THE SOFTWARE IS PROVIDED "AS IS", WITHOUT WARRANTY OF ANY KIND, EXPRESS OR 
IMPLIED, INCLUDING BUT NOT LIMITED TO THE WARRANTIES OF MERCHANTABILITY, 
FITNESS FOR A PARTICULAR PURPOSE AND NONINFRINGEMENT. IN NO EVENT SHALL THE 
AUTHORS OR COPYRIGHT HOLDERS BE LIABLE FOR ANY CLAIM, DAMAGES OR OTHER 
LIABILITY, WHETHER IN AN ACTION OF CONTRACT, TORT OR OTHERWISE, ARISING FROM, 
OUT OF OR IN CONNECTION WITH THE SOFTWARE OR THE USE OR OTHER DEALINGS 
IN THE SOFTWARE.
*)
fin := FALSE;
                    
END_ACTION
END_PROGRAM

(* Moves VG in x, y and z axis Copyright (c) 2019 Manuel Goester, Michael Witt, Klaus Kammerer Institute of Databases and Information Systems, Ulm University, Germany Permission is hereby granted, free of charge, to any person obtaining a copy of this software and associated documentation files (the "Software"), to deal in the Software without restriction, including without limitation the rights to use, copy, modify, merge, publish, distribute, sublicense, and/or sell copies of the Software, and to permit persons to whom the Software is furnished to do so, subject to the following conditions: The above copyright notice and this permission notice shall be included in all copies or substantial portions of the Software. THE SOFTWARE IS PROVIDED "AS IS", WITHOUT WARRANTY OF ANY KIND, EXPRESS OR IMPLIED, INCLUDING BUT NOT LIMITED TO THE WARRANTIES OF MERCHANTABILITY, FITNESS FOR A PARTICULAR PURPOSE AND NONINFRINGEMENT. IN NO EVENT SHALL THE AUTHORS OR COPYRIGHT HOLDERS BE LIABLE FOR ANY CLAIM, DAMAGES OR OTHER LIABILITY, WHETHER IN AN ACTION OF CONTRACT, TORT OR OTHERWISE, ARISING FROM, OUT OF OR IN CONNECTION WITH THE SOFTWARE OR THE USE OR OTHER DEALINGS IN THE SOFTWARE. *)
FUNCTION_BLOCK VG_MOVE
  VAR_INPUT
    x : INT;  (* distance VG will go forward (positive value) or backward (negative value) *)
    y : INT;  (* distance VG will go down (positive value) or up (negative value) *)
    z : INT;  (* distance VG will go counter clockwise (positive value) or clockwise (negative value) *)
  END_VAR
  VAR
    xFin : BOOL := FALSE;  (* finish flags *)
    yFin : BOOL := FALSE;
    zFin : BOOL := FALSE;
    fin : BOOL := FALSE;
    xAlreadyCounted : BOOL := FALSE;  (* true, if an impulse coming from the motor has been already counted *)
    yAlreadyCounted : BOOL := FALSE;
    zAlreadyCounted : BOOL := FALSE;
    cX : INT := 0;  (* counters *)
    cY : INT := 0;
    cZ : INT := 0;
  END_VAR

                  fin := FALSE;

// X AXIS (Forward/Backward)
IF x < 0 THEN
	// drive backward
	IF cX = x THEN
		// if counter reached demanded position, we're done
		VG.mHorizontalBackward := FALSE;
		xFin := TRUE;
	ELSE
		xFin := FALSE;
		IF cX > x THEN
			VG.mHorizontalBackward := TRUE;
			IF VG.encHorizontal AND NOT(xAlreadyCounted) THEN
				// update local counter
				cX := cX - 1;
				// update global counter
				VG.cX := VG.cX - 1;
				xAlreadyCounted := TRUE;
			ELSIF NOT(VG.encHorizontal) THEN
				xAlreadyCounted := FALSE;
			END_IF
		END_IF
	END_IF
ELSE
	// x >= 0
	// drive forward
	IF cX = x THEN
		// if counter reached demanded position, we're done
		VG.mHorizontalForward := FALSE;
		xFin := TRUE;
	ELSE
		xFin := FALSE;
		IF cX < x THEN
			VG.mHorizontalForward := TRUE;
			IF VG.encHorizontal AND NOT(xAlreadyCounted) THEN
				// update local counter
				cX := cX + 1;
				// update global counter
				VG.cX := VG.cX + 1;
				xAlreadyCounted := TRUE;
			ELSIF NOT(VG.encHorizontal) THEN
				xAlreadyCounted := FALSE;
			END_IF
		END_IF
	END_IF
END_IF

// Y AXIS (Up/Down)
IF y < 0 THEN
	// drive up
	IF cY = y THEN
		// if counter reached demanded position, we're done
		VG.mVerticalUp := FALSE;
		yFin := TRUE;
	ELSE
		yFin := FALSE;
		IF cY > y THEN
			VG.mVerticalUp := TRUE;
			IF VG.encVertical AND NOT(yAlreadyCounted) THEN
				// update local counter
				cY := cY - 1;
				// update global counter
				VG.cY := VG.cY - 1;
				yAlreadyCounted := TRUE;
			ELSIF NOT(VG.encVertical) THEN
				yAlreadyCounted := FALSE;
			END_IF
		END_IF
	END_IF
ELSE
	// y >= 0
	// drive down
	IF cY = y THEN
		// if counter reached demanded position, we're done
		VG.mVerticalDown := FALSE;
	yFin := TRUE;
	ELSE
		yFin := FALSE;
		IF cY < y THEN
			VG.mVerticalDown := TRUE;
			IF VG.encVertical AND NOT(yAlreadyCounted) THEN
				// update local counter
				cY := cY + 1;
				// update global counter
				VG.cY := VG.cY + 1;
				yAlreadyCounted := TRUE;
			ELSIF NOT(VG.encVertical) THEN
				yAlreadyCounted := FALSE;
			END_IF
		END_IF
	END_IF
END_IF

// Z AXIS (Rotation)
IF z < 0 THEN
	// drive clockwise
	IF cZ = z THEN
		// if counter reached demanded position, we're done
		VG.mRotationClockwise := FALSE;
		zFin := TRUE;
	ELSE
		zFin := FALSE;
		IF cZ > z THEN
			VG.mRotationClockwise := TRUE;
			IF VG.encRotation AND NOT(zAlreadyCounted) THEN
				// update local counter
				cZ := cZ - 1;
				// update global counter
				VG.cZ := VG.cZ - 1;
				zAlreadyCounted := TRUE;
			ELSIF NOT(VG.encRotation) THEN
				zAlreadyCounted := FALSE;
			END_IF
		END_IF
	END_IF
ELSE
	// z >= 0
	// drive counter clockwise
	IF cZ = z THEN
		// if counter reached demanded position, we're done
		VG.mRotationCClockwise := FALSE;
		zFin := TRUE;
	ELSE
		zFin := FALSE;
		IF cZ < z THEN
			VG.mRotationCClockwise := TRUE;
			IF VG.encRotation AND NOT(zAlreadyCounted) THEN
				// update local counter
				cZ := cZ + 1;
				// update global counter
				VG.cZ := VG.cZ + 1;
				zAlreadyCounted := TRUE;
			ELSIF NOT(VG.encRotation) THEN
				zAlreadyCounted := FALSE;
			END_IF
		END_IF
	END_IF
END_IF

// if all axes are finsihed, we're done
IF xFin AND yFin AND zFin THEN
	// reset local counters
	cX := 0;
	cY := 0;
	cZ := 0;
	fin := TRUE;
	RETURN;
END_IF
                
END_FUNCTION_BLOCK

PROGRAM HR_MULTI_MODE
  VAR
    fin : BOOL;
    hr_get : HR_GET_W;
    hr_store : HR_STORE_W;
    hr_put_w_on_conveyor : HR_PUT_W_ON_CONVEYOR;
    calibrateYAxis : INT := 0;  (* for GET_W calibrate y axis of rack every 3th workpiece *)
    calibarteYAxisCounted : BOOL := FALSE;
    step : INT := 1;
    timer : TON;
  END_VAR

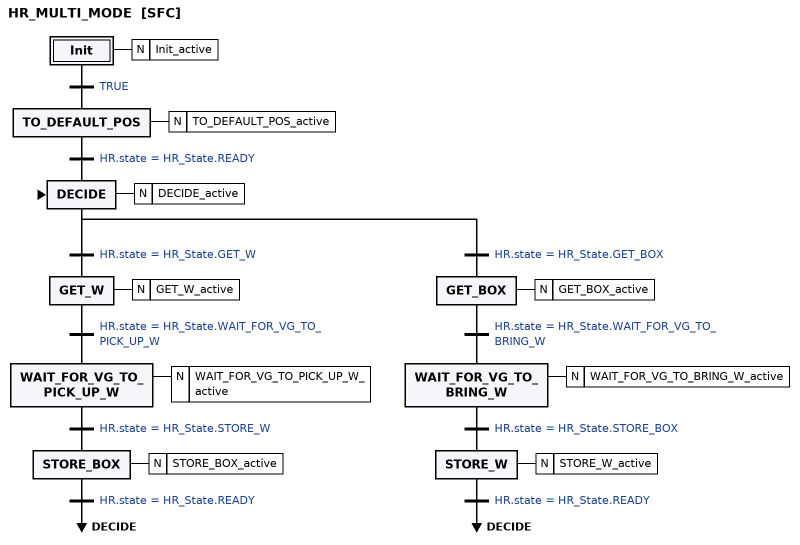
INITIAL_STEP Init:
  Init_active(N);
END_STEP
TRANSITION FROM Init TO TO_DEFAULT_POS
  := TRUE;
END_TRANSITION
STEP TO_DEFAULT_POS:
  TO_DEFAULT_POS_active(N);
END_STEP
TRANSITION FROM TO_DEFAULT_POS TO DECIDE
  := HR.state = HR_State.READY;
END_TRANSITION
STEP DECIDE:
  DECIDE_active(N);
END_STEP
TRANSITION FROM DECIDE TO GET_W
  := HR.state = HR_State.GET_W;
END_TRANSITION
TRANSITION FROM DECIDE TO GET_BOX
  := HR.state = HR_State.GET_BOX;
END_TRANSITION
STEP GET_W:
  GET_W_active(N);
END_STEP
TRANSITION FROM GET_W TO WAIT_FOR_VG_TO_PICK_UP_W
  := HR.state = HR_State.WAIT_FOR_VG_TO_PICK_UP_W;
END_TRANSITION
STEP WAIT_FOR_VG_TO_PICK_UP_W:
  WAIT_FOR_VG_TO_PICK_UP_W_active(N);
END_STEP
TRANSITION FROM WAIT_FOR_VG_TO_PICK_UP_W TO STORE_BOX
  := HR.state = HR_State.STORE_W;
END_TRANSITION
STEP STORE_BOX:
  STORE_BOX_active(N);
END_STEP
TRANSITION FROM STORE_BOX TO DECIDE
  := HR.state = HR_State.READY;
END_TRANSITION
STEP GET_BOX:
  GET_BOX_active(N);
END_STEP
TRANSITION FROM GET_BOX TO WAIT_FOR_VG_TO_BRING_W
  := HR.state = HR_State.WAIT_FOR_VG_TO_BRING_W;
END_TRANSITION
STEP WAIT_FOR_VG_TO_BRING_W:
  WAIT_FOR_VG_TO_BRING_W_active(N);
END_STEP
TRANSITION FROM WAIT_FOR_VG_TO_BRING_W TO STORE_W
  := HR.state = HR_State.STORE_BOX;
END_TRANSITION
STEP STORE_W:
  STORE_W_active(N);
END_STEP
TRANSITION FROM STORE_W TO DECIDE
  := HR.state = HR_State.READY;
END_TRANSITION

ACTION STORE_BOX_active:
                      (*
Copyright (c) 2019 Manuel Goester, Michael Witt, Klaus Kammerer
Institute of Databases and Information Systems, Ulm University, Germany

Permission is hereby granted, free of charge, to any person obtaining a copy 
of this software and associated documentation files (the "Software"), to deal 
in the Software without restriction, including without limitation the rights 
to use, copy, modify, merge, publish, distribute, sublicense, and/or sell 
copies of the Software, and to permit persons to whom the Software is 
furnished to do so, subject to the following conditions:

The above copyright notice and this permission notice shall be included in 
all copies or substantial portions of the Software.

THE SOFTWARE IS PROVIDED "AS IS", WITHOUT WARRANTY OF ANY KIND, EXPRESS OR 
IMPLIED, INCLUDING BUT NOT LIMITED TO THE WARRANTIES OF MERCHANTABILITY, 
FITNESS FOR A PARTICULAR PURPOSE AND NONINFRINGEMENT. IN NO EVENT SHALL THE 
AUTHORS OR COPYRIGHT HOLDERS BE LIABLE FOR ANY CLAIM, DAMAGES OR OTHER 
LIABILITY, WHETHER IN AN ACTION OF CONTRACT, TORT OR OTHERWISE, ARISING FROM, 
OUT OF OR IN CONNECTION WITH THE SOFTWARE OR THE USE OR OTHER DEALINGS 
IN THE SOFTWARE.
*)
IF NOT fin THEN
	// store box in rack
	hr_store(w := HR.currW);
	fin := hr_store.fin;
ELSE
	fin := FALSE;
	HR.state := HR_State.READY;
END_IF
                    
END_ACTION

ACTION GET_W_active:
                      (*
Copyright (c) 2019 Manuel Goester, Michael Witt, Klaus Kammerer
Institute of Databases and Information Systems, Ulm University, Germany

Permission is hereby granted, free of charge, to any person obtaining a copy 
of this software and associated documentation files (the "Software"), to deal 
in the Software without restriction, including without limitation the rights 
to use, copy, modify, merge, publish, distribute, sublicense, and/or sell 
copies of the Software, and to permit persons to whom the Software is 
furnished to do so, subject to the following conditions:

The above copyright notice and this permission notice shall be included in 
all copies or substantial portions of the Software.

THE SOFTWARE IS PROVIDED "AS IS", WITHOUT WARRANTY OF ANY KIND, EXPRESS OR 
IMPLIED, INCLUDING BUT NOT LIMITED TO THE WARRANTIES OF MERCHANTABILITY, 
FITNESS FOR A PARTICULAR PURPOSE AND NONINFRINGEMENT. IN NO EVENT SHALL THE 
AUTHORS OR COPYRIGHT HOLDERS BE LIABLE FOR ANY CLAIM, DAMAGES OR OTHER 
LIABILITY, WHETHER IN AN ACTION OF CONTRACT, TORT OR OTHERWISE, ARISING FROM, 
OUT OF OR IN CONNECTION WITH THE SOFTWARE OR THE USE OR OTHER DEALINGS 
IN THE SOFTWARE.
*)
// increment y calibration counter
IF NOT(calibarteYAxisCounted) THEN
	calibrateYAxis := calibrateYAxis + 1;
	calibarteYAxisCounted := TRUE;
END_IF

IF calibrateYAxis >= 3 THEN
	// calibrate y axis
	IF NOT(HR.sVertical) THEN
		HR.mVerticalUp := TRUE;
	ELSE
		Hr.mVerticalUp := FALSE;
		Hr.cY := 0;
		calibrateYAxis := 0;
	END_IF
ELSE
	CASE step OF
		1:
			// get w from rack
			IF NOT fin THEN
				hr_get(w:= HR.currW);
				fin := hr_get.fin;
			ELSE
				fin := FALSE;
				step := step + 1;
			END_IF
		2:
			// put w on conveyor
			hr_put_w_on_conveyor(w := HR.currW);
			fin := hr_put_w_on_conveyor.fin;	
			IF fin THEN
				step := step + 1;
				fin := FALSE;
			END_IF
		3:
			// bring it to VG in conveyor
			IF HR.lbOut THEN
				HR.mCbForward := TRUE;
			ELSE
				// start 1 sec timer to drive conveyor 1 sec longer to be sure that box is at outside pos
				timer(IN:= TRUE, PT := T#1S);
				IF NOT(timer.Q = FALSE AND timer.IN) THEN
					timer(IN:= FALSE);
					HR.mCbForward := FALSE;
					step := step + 1; 
				END_IF
			END_IF
		4:
			// finished
			step := 1;
			HR.state := HR_State.WAIT_FOR_VG_TO_PICK_UP_W;
			calibarteYAxisCounted := FALSE;
			// bend VG pointers to current workpiece of HR
			VG.bIdx := TC.currBatchJobIdx;
			VG.wIdx := TC.batchJobQueue.batchJobs[TC.currBatchJobIdx].nextNotProcessedIdx;
			VG.currW := TC.batchJobQueue.batchJobs[VG.bIdx].workpieces[VG.wIdx];
	END_CASE
END_IF


                    
END_ACTION

ACTION WAIT_FOR_VG_TO_PICK_UP_W_active:
                      (*
Copyright (c) 2019 Manuel Goester, Michael Witt, Klaus Kammerer
Institute of Databases and Information Systems, Ulm University, Germany

Permission is hereby granted, free of charge, to any person obtaining a copy 
of this software and associated documentation files (the "Software"), to deal 
in the Software without restriction, including without limitation the rights 
to use, copy, modify, merge, publish, distribute, sublicense, and/or sell 
copies of the Software, and to permit persons to whom the Software is 
furnished to do so, subject to the following conditions:

The above copyright notice and this permission notice shall be included in 
all copies or substantial portions of the Software.

THE SOFTWARE IS PROVIDED "AS IS", WITHOUT WARRANTY OF ANY KIND, EXPRESS OR 
IMPLIED, INCLUDING BUT NOT LIMITED TO THE WARRANTIES OF MERCHANTABILITY, 
FITNESS FOR A PARTICULAR PURPOSE AND NONINFRINGEMENT. IN NO EVENT SHALL THE 
AUTHORS OR COPYRIGHT HOLDERS BE LIABLE FOR ANY CLAIM, DAMAGES OR OTHER 
LIABILITY, WHETHER IN AN ACTION OF CONTRACT, TORT OR OTHERWISE, ARISING FROM, 
OUT OF OR IN CONNECTION WITH THE SOFTWARE OR THE USE OR OTHER DEALINGS 
IN THE SOFTWARE.
*)
IF VG.state = VG_State.TO_FUR_PUT_W OR VG.state = VG_State.TO_EJECT THEN
	HR.state := HR_State.STORE_W;
	HR.decidedToTakeANewW := FALSE;
END_IF
                    
END_ACTION

ACTION GET_BOX_active:
                      (*
Copyright (c) 2019 Manuel Goester, Michael Witt, Klaus Kammerer
Institute of Databases and Information Systems, Ulm University, Germany

Permission is hereby granted, free of charge, to any person obtaining a copy 
of this software and associated documentation files (the "Software"), to deal 
in the Software without restriction, including without limitation the rights 
to use, copy, modify, merge, publish, distribute, sublicense, and/or sell 
copies of the Software, and to permit persons to whom the Software is 
furnished to do so, subject to the following conditions:

The above copyright notice and this permission notice shall be included in 
all copies or substantial portions of the Software.

THE SOFTWARE IS PROVIDED "AS IS", WITHOUT WARRANTY OF ANY KIND, EXPRESS OR 
IMPLIED, INCLUDING BUT NOT LIMITED TO THE WARRANTIES OF MERCHANTABILITY, 
FITNESS FOR A PARTICULAR PURPOSE AND NONINFRINGEMENT. IN NO EVENT SHALL THE 
AUTHORS OR COPYRIGHT HOLDERS BE LIABLE FOR ANY CLAIM, DAMAGES OR OTHER 
LIABILITY, WHETHER IN AN ACTION OF CONTRACT, TORT OR OTHERWISE, ARISING FROM, 
OUT OF OR IN CONNECTION WITH THE SOFTWARE OR THE USE OR OTHER DEALINGS 
IN THE SOFTWARE.
*)
CASE step OF
	1:
		IF NOT fin THEN
			hr_get(w:= HR.currW);
			fin := hr_get.fin;
		ELSE
			step := step + 1;
			fin := FALSE;
		END_IF
	2:
		// put w on conveyor
		hr_put_w_on_conveyor(w := HR.currW);
		fin := hr_put_w_on_conveyor.fin;	
		IF fin THEN
			step := step + 1;
			fin := FALSE;
		END_IF
	3:
		// bring it to VG in conveyor
		IF HR.lbOut THEN
			HR.mCbForward := TRUE;
		ELSE
			// start 1 sec timer to drive conveyor 1 sec longer to be sure that box is at outside pos
			timer(IN:= TRUE, PT := T#1S);
			IF NOT(timer.Q = FALSE AND timer.IN) THEN
				timer(IN:= FALSE);
				HR.mCbForward := FALSE;
				step := step + 1; 
			END_IF
		END_IF
	4:
		// finished
		step := 1;
		HR.state := HR_State.WAIT_FOR_VG_TO_BRING_W;
END_CASE
                    
END_ACTION

ACTION DECIDE_active:
                      (*
Copyright (c) 2019 Manuel Goester, Michael Witt, Klaus Kammerer
Institute of Databases and Information Systems, Ulm University, Germany

Permission is hereby granted, free of charge, to any person obtaining a copy 
of this software and associated documentation files (the "Software"), to deal 
in the Software without restriction, including without limitation the rights 
to use, copy, modify, merge, publish, distribute, sublicense, and/or sell 
copies of the Software, and to permit persons to whom the Software is 
furnished to do so, subject to the following conditions:

The above copyright notice and this permission notice shall be included in 
all copies or substantial portions of the Software.

THE SOFTWARE IS PROVIDED "AS IS", WITHOUT WARRANTY OF ANY KIND, EXPRESS OR 
IMPLIED, INCLUDING BUT NOT LIMITED TO THE WARRANTIES OF MERCHANTABILITY, 
FITNESS FOR A PARTICULAR PURPOSE AND NONINFRINGEMENT. IN NO EVENT SHALL THE 
AUTHORS OR COPYRIGHT HOLDERS BE LIABLE FOR ANY CLAIM, DAMAGES OR OTHER 
LIABILITY, WHETHER IN AN ACTION OF CONTRACT, TORT OR OTHERWISE, ARISING FROM, 
OUT OF OR IN CONNECTION WITH THE SOFTWARE OR THE USE OR OTHER DEALINGS 
IN THE SOFTWARE.
*)

// if sl positions free or if not free if workpiece will not be ejected 
// AND VG is not storing
// AND HR does not already decided to take a new workpiece
// THEN 
IF ((SL.lbRed AND SL.lbWhite AND SL.lbBlue) OR (SL.currW.format.ejectEnabled AND NOT(SL.currW.state = W_State.NULL))) AND NOT(VG.storeW) AND NOT(decidedToTakeANewW) THEN
	HR.bIdx := 0;
	HR.wIdx := 0;
	HR.currW := TC.nullW;
	HR.decidedToTakeANewW := TRUE;
	VG.storeW := FALSE;
ELSIF HR.decidedToTakeANewW THEN
	// get new w out of rack
	IF TC.state = TC_state.W_LOADED THEN
		// set pointers to make sure that they are set
		Hr.bIdx := TC.currBatchJobIdx;
		Hr.wIdx := TC.batchJobQueue.batchJobs[TC.currBatchJobIdx].nextNotProcessedIdx;
		HR.currW := TC.batchJobQueue.batchJobs[Hr.bIdx].workpieces[Hr.wIdx];
		// workpiece is loaded, start production
		HR.state := HR_State.GET_W;
		// signalise that production starts
		TC.state := TC_State.WAIT_UNTIL_W_FINISHED;
	ELSE
		// no workpiece loaded, load it now
		TC.state := TC_State.LOAD_NEXT_W;
	END_IF
ELSE
	// prevent misconduct when a workpiece is still lying in one of the three spots at SL, although the application got reset
	IF NOT(VG.bIdx = 0) THEN
		// get empty box out of rack
		// set workpiece to get the right box from rack
		IF NOT(SL.lbWhite) OR NOT(SL.lbRed) OR NOT(SL.lbBlue) THEN
			HR.bIdx := SL.bIdx;
			HR.wIdx := SL.wIdx;
			HR.currW := SL.currW;
		ELSE
			HR.bIdx := VG.bIdx;
			HR.wIdx := VG.wIdx;
			HR.currW := VG.currW;
		END_IF
		HR.state := HR_State.GET_BOX;
		// reset flag
		VG.storeW := FALSE;
		END_IF
END_IF
                    
END_ACTION

ACTION STORE_W_active:
                      (*
Copyright (c) 2019 Manuel Goester, Michael Witt, Klaus Kammerer
Institute of Databases and Information Systems, Ulm University, Germany

Permission is hereby granted, free of charge, to any person obtaining a copy 
of this software and associated documentation files (the "Software"), to deal 
in the Software without restriction, including without limitation the rights 
to use, copy, modify, merge, publish, distribute, sublicense, and/or sell 
copies of the Software, and to permit persons to whom the Software is 
furnished to do so, subject to the following conditions:

The above copyright notice and this permission notice shall be included in 
all copies or substantial portions of the Software.

THE SOFTWARE IS PROVIDED "AS IS", WITHOUT WARRANTY OF ANY KIND, EXPRESS OR 
IMPLIED, INCLUDING BUT NOT LIMITED TO THE WARRANTIES OF MERCHANTABILITY, 
FITNESS FOR A PARTICULAR PURPOSE AND NONINFRINGEMENT. IN NO EVENT SHALL THE 
AUTHORS OR COPYRIGHT HOLDERS BE LIABLE FOR ANY CLAIM, DAMAGES OR OTHER 
LIABILITY, WHETHER IN AN ACTION OF CONTRACT, TORT OR OTHERWISE, ARISING FROM, 
OUT OF OR IN CONNECTION WITH THE SOFTWARE OR THE USE OR OTHER DEALINGS 
IN THE SOFTWARE.
*)
IF NOT fin THEN
	// store workpiece in rack
	hr_store(w := HR.currW);
	fin := hr_store.fin;
ELSE
	fin := FALSE;
	HR.state := HR_State.READY;
END_IF
                    
END_ACTION

ACTION WAIT_FOR_VG_TO_BRING_W_active:
                      (*
Copyright (c) 2019 Manuel Goester, Michael Witt, Klaus Kammerer
Institute of Databases and Information Systems, Ulm University, Germany

Permission is hereby granted, free of charge, to any person obtaining a copy 
of this software and associated documentation files (the "Software"), to deal 
in the Software without restriction, including without limitation the rights 
to use, copy, modify, merge, publish, distribute, sublicense, and/or sell 
copies of the Software, and to permit persons to whom the Software is 
furnished to do so, subject to the following conditions:

The above copyright notice and this permission notice shall be included in 
all copies or substantial portions of the Software.

THE SOFTWARE IS PROVIDED "AS IS", WITHOUT WARRANTY OF ANY KIND, EXPRESS OR 
IMPLIED, INCLUDING BUT NOT LIMITED TO THE WARRANTIES OF MERCHANTABILITY, 
FITNESS FOR A PARTICULAR PURPOSE AND NONINFRINGEMENT. IN NO EVENT SHALL THE 
AUTHORS OR COPYRIGHT HOLDERS BE LIABLE FOR ANY CLAIM, DAMAGES OR OTHER 
LIABILITY, WHETHER IN AN ACTION OF CONTRACT, TORT OR OTHERWISE, ARISING FROM, 
OUT OF OR IN CONNECTION WITH THE SOFTWARE OR THE USE OR OTHER DEALINGS 
IN THE SOFTWARE.
*)
IF VG.state = VG_State.TO_HR_PUT_W_FINISHED OR HR.currW.format.ejectEnabled THEN
	HR.state := HR_State.STORE_BOX;
END_IF
                    
END_ACTION

ACTION Init_active:
                      (*
Copyright (c) 2019 Manuel Goester, Michael Witt, Klaus Kammerer
Institute of Databases and Information Systems, Ulm University, Germany

Permission is hereby granted, free of charge, to any person obtaining a copy 
of this software and associated documentation files (the "Software"), to deal 
in the Software without restriction, including without limitation the rights 
to use, copy, modify, merge, publish, distribute, sublicense, and/or sell 
copies of the Software, and to permit persons to whom the Software is 
furnished to do so, subject to the following conditions:

The above copyright notice and this permission notice shall be included in 
all copies or substantial portions of the Software.

THE SOFTWARE IS PROVIDED "AS IS", WITHOUT WARRANTY OF ANY KIND, EXPRESS OR 
IMPLIED, INCLUDING BUT NOT LIMITED TO THE WARRANTIES OF MERCHANTABILITY, 
FITNESS FOR A PARTICULAR PURPOSE AND NONINFRINGEMENT. IN NO EVENT SHALL THE 
AUTHORS OR COPYRIGHT HOLDERS BE LIABLE FOR ANY CLAIM, DAMAGES OR OTHER 
LIABILITY, WHETHER IN AN ACTION OF CONTRACT, TORT OR OTHERWISE, ARISING FROM, 
OUT OF OR IN CONNECTION WITH THE SOFTWARE OR THE USE OR OTHER DEALINGS 
IN THE SOFTWARE.
*)
calibrateYAxis := 0;
calibarteYAxisCounted := FALSE;
                    
END_ACTION

ACTION TO_DEFAULT_POS_active:
                      (*
Copyright (c) 2019 Manuel Goester, Michael Witt, Klaus Kammerer
Institute of Databases and Information Systems, Ulm University, Germany

Permission is hereby granted, free of charge, to any person obtaining a copy 
of this software and associated documentation files (the "Software"), to deal 
in the Software without restriction, including without limitation the rights 
to use, copy, modify, merge, publish, distribute, sublicense, and/or sell 
copies of the Software, and to permit persons to whom the Software is 
furnished to do so, subject to the following conditions:

The above copyright notice and this permission notice shall be included in 
all copies or substantial portions of the Software.

THE SOFTWARE IS PROVIDED "AS IS", WITHOUT WARRANTY OF ANY KIND, EXPRESS OR 
IMPLIED, INCLUDING BUT NOT LIMITED TO THE WARRANTIES OF MERCHANTABILITY, 
FITNESS FOR A PARTICULAR PURPOSE AND NONINFRINGEMENT. IN NO EVENT SHALL THE 
AUTHORS OR COPYRIGHT HOLDERS BE LIABLE FOR ANY CLAIM, DAMAGES OR OTHER 
LIABILITY, WHETHER IN AN ACTION OF CONTRACT, TORT OR OTHERWISE, ARISING FROM, 
OUT OF OR IN CONNECTION WITH THE SOFTWARE OR THE USE OR OTHER DEALINGS 
IN THE SOFTWARE.
*)
// returns High Rack TOWER to its default start position
// set "ausleger" arm to default position
IF HR.sCBack = FALSE THEN
	HR.mCBackward := TRUE;
ELSE 
	HR.mCBackward := FALSE;
	// set tower vertical position to max UP as well as horizontal position max RIGHT
	IF HR.sHorizontal = FALSE THEN
		HR.mHorizontalRight := TRUE;
	ELSE
		HR.mHorizontalRight := FALSE;
	END_IF
	
	IF HR.sVertical = FALSE THEN
		HR.mVerticalUp := TRUE;
	ELSE
		HR.mVerticalUp := FALSE;
	END_IF
END_IF

IF HR.sHorizontal AND HR.sVertical AND HR.sCBack THEN
	HR.cX := 0;
	HR.cY := 0;
	HR.state := HR_State.READY;
END_IF
                    
END_ACTION
END_PROGRAM

(* Constructor for Format A Format defines the options for a production of a workpiece Copyright (c) 2019 Manuel Goester, Michael Witt, Klaus Kammerer Institute of Databases and Information Systems, Ulm University, Germany Permission is hereby granted, free of charge, to any person obtaining a copy of this software and associated documentation files (the "Software"), to deal in the Software without restriction, including without limitation the rights to use, copy, modify, merge, publish, distribute, sublicense, and/or sell copies of the Software, and to permit persons to whom the Software is furnished to do so, subject to the following conditions: The above copyright notice and this permission notice shall be included in all copies or substantial portions of the Software. THE SOFTWARE IS PROVIDED "AS IS", WITHOUT WARRANTY OF ANY KIND, EXPRESS OR IMPLIED, INCLUDING BUT NOT LIMITED TO THE WARRANTIES OF MERCHANTABILITY, FITNESS FOR A PARTICULAR PURPOSE AND NONINFRINGEMENT. IN NO EVENT SHALL THE AUTHORS OR COPYRIGHT HOLDERS BE LIABLE FOR ANY CLAIM, DAMAGES OR OTHER LIABILITY, WHETHER IN AN ACTION OF CONTRACT, TORT OR OTHERWISE, ARISING FROM, OUT OF OR IN CONNECTION WITH THE SOFTWARE OR THE USE OR OTHER DEALINGS IN THE SOFTWARE. *)
FUNCTION newFormat : Format
  VAR_INPUT
    furEnabled : BOOL;
    sawEnabled : BOOL;
    colorCheckEnabled : BOOL;
    ejectEnabled : BOOL;
    furDuration : TIME;
    sawDuration : TIME;
  END_VAR

                  newFormat.furEnabled := furEnabled;
newFormat.sawEnabled := sawEnabled;
newFormat.colorCheckEnabled := colorCheckEnabled;
newFormat.ejectEnabled := ejectEnabled;
newFormat.furDuration := furDuration;
newFormat.sawDuration := sawDuration;
RETURN;
                
END_FUNCTION

(* Constructor of a BatchJob Copyright (c) 2019 Manuel Goester, Michael Witt, Klaus Kammerer Institute of Databases and Information Systems, Ulm University, Germany Permission is hereby granted, free of charge, to any person obtaining a copy of this software and associated documentation files (the "Software"), to deal in the Software without restriction, including without limitation the rights to use, copy, modify, merge, publish, distribute, sublicense, and/or sell copies of the Software, and to permit persons to whom the Software is furnished to do so, subject to the following conditions: The above copyright notice and this permission notice shall be included in all copies or substantial portions of the Software. THE SOFTWARE IS PROVIDED "AS IS", WITHOUT WARRANTY OF ANY KIND, EXPRESS OR IMPLIED, INCLUDING BUT NOT LIMITED TO THE WARRANTIES OF MERCHANTABILITY, FITNESS FOR A PARTICULAR PURPOSE AND NONINFRINGEMENT. IN NO EVENT SHALL THE AUTHORS OR COPYRIGHT HOLDERS BE LIABLE FOR ANY CLAIM, DAMAGES OR OTHER LIABILITY, WHETHER IN AN ACTION OF CONTRACT, TORT OR OTHERWISE, ARISING FROM, OUT OF OR IN CONNECTION WITH THE SOFTWARE OR THE USE OR OTHER DEALINGS IN THE SOFTWARE. *)
FUNCTION newBatchJob : BatchJob
  VAR_INPUT
    batchSize : INT;  (* amount of workpieces in batch job *)
    workpieces : ARRAY[1..9] OF Workpiece;  (* workpieces being processed *)
    mode : ExecutionMode;  (* type of execution: single, multi or sorting *)
  END_VAR
  VAR
    placeFound : BOOL := FALSE;
    wsFull : BOOL := FALSE;
    i : INT := 1;
    sysTime : RTC;
  END_VAR

                  newBatchJob.batchSize := batchSize;
newBatchJob.workpieces := workpieces;
newBatchJob.mode := mode;

// Search for next free position in workpieces. If there is no free position, set nextFreeWPos to -1
WHILE NOT(placeFound) AND NOT(wsFull) DO
	IF workpieces[i].state = W_State.NULL THEN
		placeFound := TRUE;
		newBatchJob.nextFreeWPos := i;
	ELSIF i > newBatchJob.batchSize THEN
		wsFull := TRUE;
		newBatchJob.nextFreeWPos := -1;
	ELSE
		i := i + 1;
	END_IF
END_WHILE

newBatchJob.nextNotProcessedIdx := 1;
newBatchJob.amountFinishedW := 0;
newBatchJob.duration := T#0S;
newBatchJob.pauseDuration := T#0S;
newBatchJob.state := BatchJobState.WAITING;
// current system time
newBatchJob.timeCreated := sysTime.CDT;
RETURN;
                
END_FUNCTION

PROGRAM HR_SINGLE_MODE
  VAR
    selectionValid : BOOL;
    tX : TON;
    tY : TON;
    xFin : BOOL;
    yFin : BOOL;
    zFin : BOOL;
    conveyorBeltFin : BOOL;
    subBlockStart : BOOL;
    fin : BOOL;
    hr_get_w : HR_GET_W;
    hr_store_w : HR_STORE_W;
    hr_put_w_on_conveyor : HR_PUT_W_ON_CONVEYOR;
    calibrateYAxis : INT;
    alreadyCounted : BOOL;
    step : INT := 1;
    timer : TON;
  END_VAR

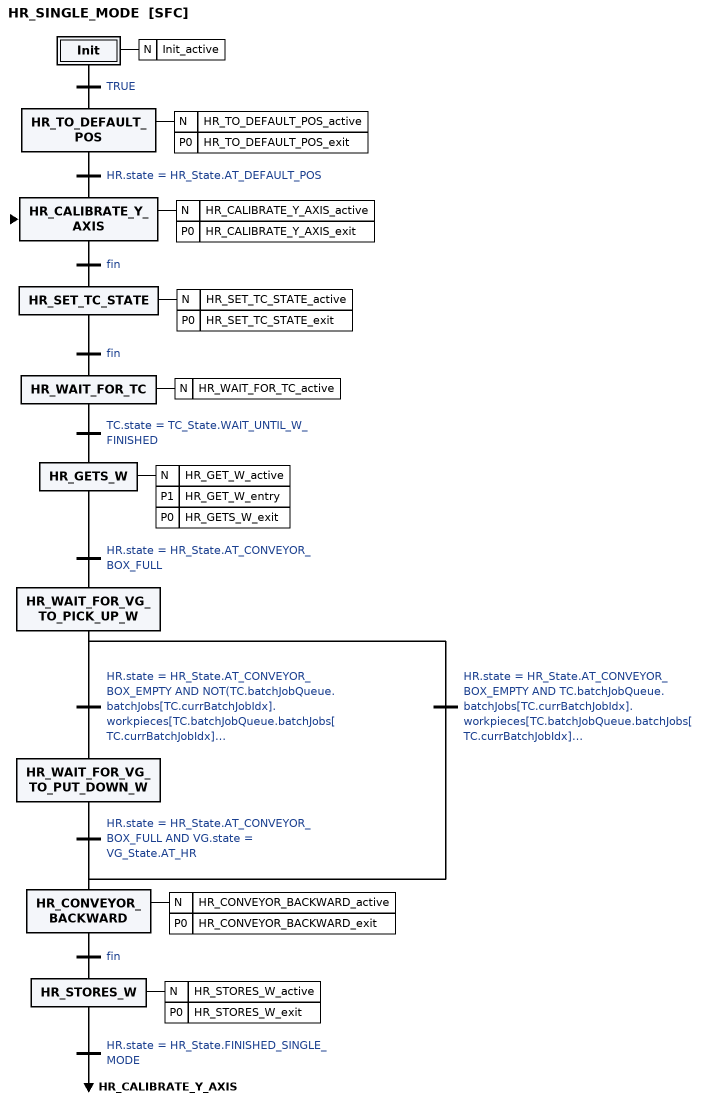
INITIAL_STEP Init:
  Init_active(N);
END_STEP
TRANSITION FROM Init TO HR_TO_DEFAULT_POS
  := TRUE;
END_TRANSITION
STEP HR_TO_DEFAULT_POS:
  HR_TO_DEFAULT_POS_active(N);
  HR_TO_DEFAULT_POS_exit(P0);
END_STEP
TRANSITION FROM HR_TO_DEFAULT_POS TO HR_CALIBRATE_Y_AXIS
  := HR.state = HR_State.AT_DEFAULT_POS;
END_TRANSITION
STEP HR_CALIBRATE_Y_AXIS:
  HR_CALIBRATE_Y_AXIS_active(N);
  HR_CALIBRATE_Y_AXIS_exit(P0);
END_STEP
TRANSITION FROM HR_CALIBRATE_Y_AXIS TO HR_SET_TC_STATE
  := fin;
END_TRANSITION
STEP HR_SET_TC_STATE:
  HR_SET_TC_STATE_active(N);
  HR_SET_TC_STATE_exit(P0);
END_STEP
TRANSITION FROM HR_SET_TC_STATE TO HR_WAIT_FOR_TC
  := fin;
END_TRANSITION
STEP HR_WAIT_FOR_TC:
  HR_WAIT_FOR_TC_active(N);
END_STEP
TRANSITION FROM HR_WAIT_FOR_TC TO HR_GETS_W
  := TC.state = TC_State.WAIT_UNTIL_W_FINISHED;
END_TRANSITION
STEP HR_GETS_W:
  HR_GET_W_active(N);
  HR_GET_W_entry(P1);
  HR_GETS_W_exit(P0);
END_STEP
TRANSITION FROM HR_GETS_W TO HR_WAIT_FOR_VG_TO_PICK_UP_W
  := HR.state = HR_State.AT_CONVEYOR_BOX_FULL;
END_TRANSITION
STEP HR_WAIT_FOR_VG_TO_PICK_UP_W:
END_STEP
TRANSITION FROM HR_WAIT_FOR_VG_TO_PICK_UP_W TO HR_WAIT_FOR_VG_TO_PUT_DOWN_W
  := HR.state = HR_State.AT_CONVEYOR_BOX_EMPTY AND NOT(TC.batchJobQueue.batchJobs[TC.currBatchJobIdx].workpieces[TC.batchJobQueue.batchJobs[TC.currBatchJobIdx].nextNotProcessedIdx].format.ejectEnabled);
END_TRANSITION
TRANSITION FROM HR_WAIT_FOR_VG_TO_PICK_UP_W TO HR_CONVEYOR_BACKWARD
  := HR.state = HR_State.AT_CONVEYOR_BOX_EMPTY AND TC.batchJobQueue.batchJobs[TC.currBatchJobIdx].workpieces[TC.batchJobQueue.batchJobs[TC.currBatchJobIdx].nextNotProcessedIdx].format.ejectEnabled;
END_TRANSITION
STEP HR_WAIT_FOR_VG_TO_PUT_DOWN_W:
END_STEP
TRANSITION FROM HR_WAIT_FOR_VG_TO_PUT_DOWN_W TO HR_CONVEYOR_BACKWARD
  := HR.state = HR_State.AT_CONVEYOR_BOX_FULL AND VG.state = VG_State.AT_HR;
END_TRANSITION
STEP HR_CONVEYOR_BACKWARD:
  HR_CONVEYOR_BACKWARD_active(N);
  HR_CONVEYOR_BACKWARD_exit(P0);
END_STEP
TRANSITION FROM HR_CONVEYOR_BACKWARD TO HR_STORES_W
  := fin;
END_TRANSITION
STEP HR_STORES_W:
  HR_STORES_W_active(N);
  HR_STORES_W_exit(P0);
END_STEP
TRANSITION FROM HR_STORES_W TO HR_CALIBRATE_Y_AXIS
  := HR.state = HR_State.FINISHED_SINGLE_MODE;
END_TRANSITION

ACTION HR_GET_W_active:
                      (*
Copyright (c) 2019 Manuel Goester, Michael Witt, Klaus Kammerer
Institute of Databases and Information Systems, Ulm University, Germany

Permission is hereby granted, free of charge, to any person obtaining a copy 
of this software and associated documentation files (the "Software"), to deal 
in the Software without restriction, including without limitation the rights 
to use, copy, modify, merge, publish, distribute, sublicense, and/or sell 
copies of the Software, and to permit persons to whom the Software is 
furnished to do so, subject to the following conditions:

The above copyright notice and this permission notice shall be included in 
all copies or substantial portions of the Software.

THE SOFTWARE IS PROVIDED "AS IS", WITHOUT WARRANTY OF ANY KIND, EXPRESS OR 
IMPLIED, INCLUDING BUT NOT LIMITED TO THE WARRANTIES OF MERCHANTABILITY, 
FITNESS FOR A PARTICULAR PURPOSE AND NONINFRINGEMENT. IN NO EVENT SHALL THE 
AUTHORS OR COPYRIGHT HOLDERS BE LIABLE FOR ANY CLAIM, DAMAGES OR OTHER 
LIABILITY, WHETHER IN AN ACTION OF CONTRACT, TORT OR OTHERWISE, ARISING FROM, 
OUT OF OR IN CONNECTION WITH THE SOFTWARE OR THE USE OR OTHER DEALINGS 
IN THE SOFTWARE.
*)
CASE step OF
	1:
		// get w from rack
		IF NOT fin THEN
			hr_get_w(w:=TC.batchJobQueue.batchJobs[TC.currBatchJobIdx].workpieces[TC.batchJobQueue.batchJobs[TC.currBatchJobIdx].nextNotProcessedIdx]);
			fin := hr_get_w.fin;
		ELSE
			fin := FALSE;
			step := step + 1;
			
		END_IF
	2:
		// put w on conveyor
		hr_put_w_on_conveyor(w := HR.currW);
		fin := hr_put_w_on_conveyor.fin;	
		IF fin THEN
			step := step + 1;
			fin := FALSE;
		END_IF
	3:
		// bring it to VG in conveyor
		IF HR.lbOut THEN
			HR.mCbForward := TRUE;
		ELSE
			// start 1 sec timer to drive conveyor 1 sec longer to be sure that box is at outside pos
			timer(IN:= TRUE, PT := T#1S);
			IF NOT(timer.Q = FALSE AND timer.IN) THEN
				timer(IN:= FALSE);
				HR.mCbForward := FALSE;
				step := step + 1; 
			END_IF
		END_IF
	4:
		// finished
		step := 1;
		HR.state := HR_State.AT_CONVEYOR_BOX_FULL;
END_CASE
                    
END_ACTION

ACTION ConveyorBack_HR_STORE_W_active_exit:
                      (*
Copyright (c) 2019 Manuel Goester, Michael Witt, Klaus Kammerer
Institute of Databases and Information Systems, Ulm University, Germany

Permission is hereby granted, free of charge, to any person obtaining a copy 
of this software and associated documentation files (the "Software"), to deal 
in the Software without restriction, including without limitation the rights 
to use, copy, modify, merge, publish, distribute, sublicense, and/or sell 
copies of the Software, and to permit persons to whom the Software is 
furnished to do so, subject to the following conditions:

The above copyright notice and this permission notice shall be included in 
all copies or substantial portions of the Software.

THE SOFTWARE IS PROVIDED "AS IS", WITHOUT WARRANTY OF ANY KIND, EXPRESS OR 
IMPLIED, INCLUDING BUT NOT LIMITED TO THE WARRANTIES OF MERCHANTABILITY, 
FITNESS FOR A PARTICULAR PURPOSE AND NONINFRINGEMENT. IN NO EVENT SHALL THE 
AUTHORS OR COPYRIGHT HOLDERS BE LIABLE FOR ANY CLAIM, DAMAGES OR OTHER 
LIABILITY, WHETHER IN AN ACTION OF CONTRACT, TORT OR OTHERWISE, ARISING FROM, 
OUT OF OR IN CONNECTION WITH THE SOFTWARE OR THE USE OR OTHER DEALINGS 
IN THE SOFTWARE.
*)
conveyorBeltFin := FALSE;
                    
END_ACTION

ACTION HR_STORES_W_active:
                      (*
Copyright (c) 2019 Manuel Goester, Michael Witt, Klaus Kammerer
Institute of Databases and Information Systems, Ulm University, Germany

Permission is hereby granted, free of charge, to any person obtaining a copy 
of this software and associated documentation files (the "Software"), to deal 
in the Software without restriction, including without limitation the rights 
to use, copy, modify, merge, publish, distribute, sublicense, and/or sell 
copies of the Software, and to permit persons to whom the Software is 
furnished to do so, subject to the following conditions:

The above copyright notice and this permission notice shall be included in 
all copies or substantial portions of the Software.

THE SOFTWARE IS PROVIDED "AS IS", WITHOUT WARRANTY OF ANY KIND, EXPRESS OR 
IMPLIED, INCLUDING BUT NOT LIMITED TO THE WARRANTIES OF MERCHANTABILITY, 
FITNESS FOR A PARTICULAR PURPOSE AND NONINFRINGEMENT. IN NO EVENT SHALL THE 
AUTHORS OR COPYRIGHT HOLDERS BE LIABLE FOR ANY CLAIM, DAMAGES OR OTHER 
LIABILITY, WHETHER IN AN ACTION OF CONTRACT, TORT OR OTHERWISE, ARISING FROM, 
OUT OF OR IN CONNECTION WITH THE SOFTWARE OR THE USE OR OTHER DEALINGS 
IN THE SOFTWARE.
*)
IF NOT fin THEN
	HR.state := HR_State.STORE_W;
	hr_store_w(w:=TC.batchJobQueue.batchJobs[TC.currBatchJobIdx].workpieces[TC.batchJobQueue.batchJobs[TC.currBatchJobIdx].nextNotProcessedIdx]);
	fin := hr_store_w.fin;
ELSIF VG.state = VG_State.AT_HR THEN
	// set BatchJobQueue to next workpiece
	HR.state := HR_State.FINISHED_SINGLE_MODE;
	// reset object
	SM.currW := TC.nullW;
	fin := FALSE;
END_IF
                    
END_ACTION

ACTION ConveyorBack_HR_STORE_W_active_active:
                      (*
Copyright (c) 2019 Manuel Goester, Michael Witt, Klaus Kammerer
Institute of Databases and Information Systems, Ulm University, Germany

Permission is hereby granted, free of charge, to any person obtaining a copy 
of this software and associated documentation files (the "Software"), to deal 
in the Software without restriction, including without limitation the rights 
to use, copy, modify, merge, publish, distribute, sublicense, and/or sell 
copies of the Software, and to permit persons to whom the Software is 
furnished to do so, subject to the following conditions:

The above copyright notice and this permission notice shall be included in 
all copies or substantial portions of the Software.

THE SOFTWARE IS PROVIDED "AS IS", WITHOUT WARRANTY OF ANY KIND, EXPRESS OR 
IMPLIED, INCLUDING BUT NOT LIMITED TO THE WARRANTIES OF MERCHANTABILITY, 
FITNESS FOR A PARTICULAR PURPOSE AND NONINFRINGEMENT. IN NO EVENT SHALL THE 
AUTHORS OR COPYRIGHT HOLDERS BE LIABLE FOR ANY CLAIM, DAMAGES OR OTHER 
LIABILITY, WHETHER IN AN ACTION OF CONTRACT, TORT OR OTHERWISE, ARISING FROM, 
OUT OF OR IN CONNECTION WITH THE SOFTWARE OR THE USE OR OTHER DEALINGS 
IN THE SOFTWARE.
*)
IF HR.lbIn THEN
	HR.mCbBackward := TRUE;
ELSE
	HR.mCbBackward := FALSE;
	conveyorBeltFin := TRUE;
END_IF
                    
END_ACTION

ACTION HR_TO_DEFAULT_POS_active:
                      (*
Copyright (c) 2019 Manuel Goester, Michael Witt, Klaus Kammerer
Institute of Databases and Information Systems, Ulm University, Germany

Permission is hereby granted, free of charge, to any person obtaining a copy 
of this software and associated documentation files (the "Software"), to deal 
in the Software without restriction, including without limitation the rights 
to use, copy, modify, merge, publish, distribute, sublicense, and/or sell 
copies of the Software, and to permit persons to whom the Software is 
furnished to do so, subject to the following conditions:

The above copyright notice and this permission notice shall be included in 
all copies or substantial portions of the Software.

THE SOFTWARE IS PROVIDED "AS IS", WITHOUT WARRANTY OF ANY KIND, EXPRESS OR 
IMPLIED, INCLUDING BUT NOT LIMITED TO THE WARRANTIES OF MERCHANTABILITY, 
FITNESS FOR A PARTICULAR PURPOSE AND NONINFRINGEMENT. IN NO EVENT SHALL THE 
AUTHORS OR COPYRIGHT HOLDERS BE LIABLE FOR ANY CLAIM, DAMAGES OR OTHER 
LIABILITY, WHETHER IN AN ACTION OF CONTRACT, TORT OR OTHERWISE, ARISING FROM, 
OUT OF OR IN CONNECTION WITH THE SOFTWARE OR THE USE OR OTHER DEALINGS 
IN THE SOFTWARE.
*)

// returns the High Rack TOWER to its default start position
// set "ausleger" arm to default position
IF HR.sCBack = FALSE THEN
	HR.mCBackward := TRUE;
ELSE 
	HR.mCBackward := FALSE;
	// set tower vertical position to max UP as well as horizontal position max RIGHT
	IF HR.sHorizontal = FALSE THEN
		HR.mHorizontalRight := TRUE;
	ELSE
		HR.mHorizontalRight := FALSE;
		HR.cX := 0;
	END_IF
	
	IF HR.sVertical = FALSE THEN
		HR.mVerticalUp := TRUE;
	ELSE
		HR.mVerticalUp := FALSE;
		HR.cY := 0;
	END_IF
END_IF

IF HR.sHorizontal AND HR.sVertical AND HR.sCBack THEN
	HR.state := HR_State.AT_DEFAULT_POS;
END_IF
                    
END_ACTION

ACTION HR_GET_W_entry:
                      (*
Copyright (c) 2019 Manuel Goester, Michael Witt, Klaus Kammerer
Institute of Databases and Information Systems, Ulm University, Germany

Permission is hereby granted, free of charge, to any person obtaining a copy 
of this software and associated documentation files (the "Software"), to deal 
in the Software without restriction, including without limitation the rights 
to use, copy, modify, merge, publish, distribute, sublicense, and/or sell 
copies of the Software, and to permit persons to whom the Software is 
furnished to do so, subject to the following conditions:

The above copyright notice and this permission notice shall be included in 
all copies or substantial portions of the Software.

THE SOFTWARE IS PROVIDED "AS IS", WITHOUT WARRANTY OF ANY KIND, EXPRESS OR 
IMPLIED, INCLUDING BUT NOT LIMITED TO THE WARRANTIES OF MERCHANTABILITY, 
FITNESS FOR A PARTICULAR PURPOSE AND NONINFRINGEMENT. IN NO EVENT SHALL THE 
AUTHORS OR COPYRIGHT HOLDERS BE LIABLE FOR ANY CLAIM, DAMAGES OR OTHER 
LIABILITY, WHETHER IN AN ACTION OF CONTRACT, TORT OR OTHERWISE, ARISING FROM, 
OUT OF OR IN CONNECTION WITH THE SOFTWARE OR THE USE OR OTHER DEALINGS 
IN THE SOFTWARE.
*)
HR.state := HR_State.GET_W;

                    
END_ACTION

ACTION HR_TO_DEFAULT_POS_exit:
                      (*
Copyright (c) 2019 Manuel Goester, Michael Witt, Klaus Kammerer
Institute of Databases and Information Systems, Ulm University, Germany

Permission is hereby granted, free of charge, to any person obtaining a copy 
of this software and associated documentation files (the "Software"), to deal 
in the Software without restriction, including without limitation the rights 
to use, copy, modify, merge, publish, distribute, sublicense, and/or sell 
copies of the Software, and to permit persons to whom the Software is 
furnished to do so, subject to the following conditions:

The above copyright notice and this permission notice shall be included in 
all copies or substantial portions of the Software.

THE SOFTWARE IS PROVIDED "AS IS", WITHOUT WARRANTY OF ANY KIND, EXPRESS OR 
IMPLIED, INCLUDING BUT NOT LIMITED TO THE WARRANTIES OF MERCHANTABILITY, 
FITNESS FOR A PARTICULAR PURPOSE AND NONINFRINGEMENT. IN NO EVENT SHALL THE 
AUTHORS OR COPYRIGHT HOLDERS BE LIABLE FOR ANY CLAIM, DAMAGES OR OTHER 
LIABILITY, WHETHER IN AN ACTION OF CONTRACT, TORT OR OTHERWISE, ARISING FROM, 
OUT OF OR IN CONNECTION WITH THE SOFTWARE OR THE USE OR OTHER DEALINGS 
IN THE SOFTWARE.
*)
HR_SINGLE_MODE.subBlockStart := FALSE;
                    
END_ACTION

ACTION HR_GETS_W_exit:
                      (*
Copyright (c) 2019 Manuel Goester, Michael Witt, Klaus Kammerer
Institute of Databases and Information Systems, Ulm University, Germany

Permission is hereby granted, free of charge, to any person obtaining a copy 
of this software and associated documentation files (the "Software"), to deal 
in the Software without restriction, including without limitation the rights 
to use, copy, modify, merge, publish, distribute, sublicense, and/or sell 
copies of the Software, and to permit persons to whom the Software is 
furnished to do so, subject to the following conditions:

The above copyright notice and this permission notice shall be included in 
all copies or substantial portions of the Software.

THE SOFTWARE IS PROVIDED "AS IS", WITHOUT WARRANTY OF ANY KIND, EXPRESS OR 
IMPLIED, INCLUDING BUT NOT LIMITED TO THE WARRANTIES OF MERCHANTABILITY, 
FITNESS FOR A PARTICULAR PURPOSE AND NONINFRINGEMENT. IN NO EVENT SHALL THE 
AUTHORS OR COPYRIGHT HOLDERS BE LIABLE FOR ANY CLAIM, DAMAGES OR OTHER 
LIABILITY, WHETHER IN AN ACTION OF CONTRACT, TORT OR OTHERWISE, ARISING FROM, 
OUT OF OR IN CONNECTION WITH THE SOFTWARE OR THE USE OR OTHER DEALINGS 
IN THE SOFTWARE.
*)
fin := FALSE;
                    
END_ACTION

ACTION HR_CONVEYOR_BACKWARD_active:
                      (*
Copyright (c) 2019 Manuel Goester, Michael Witt, Klaus Kammerer
Institute of Databases and Information Systems, Ulm University, Germany

Permission is hereby granted, free of charge, to any person obtaining a copy 
of this software and associated documentation files (the "Software"), to deal 
in the Software without restriction, including without limitation the rights 
to use, copy, modify, merge, publish, distribute, sublicense, and/or sell 
copies of the Software, and to permit persons to whom the Software is 
furnished to do so, subject to the following conditions:

The above copyright notice and this permission notice shall be included in 
all copies or substantial portions of the Software.

THE SOFTWARE IS PROVIDED "AS IS", WITHOUT WARRANTY OF ANY KIND, EXPRESS OR 
IMPLIED, INCLUDING BUT NOT LIMITED TO THE WARRANTIES OF MERCHANTABILITY, 
FITNESS FOR A PARTICULAR PURPOSE AND NONINFRINGEMENT. IN NO EVENT SHALL THE 
AUTHORS OR COPYRIGHT HOLDERS BE LIABLE FOR ANY CLAIM, DAMAGES OR OTHER 
LIABILITY, WHETHER IN AN ACTION OF CONTRACT, TORT OR OTHERWISE, ARISING FROM, 
OUT OF OR IN CONNECTION WITH THE SOFTWARE OR THE USE OR OTHER DEALINGS 
IN THE SOFTWARE.
*)
IF HR.lbIn THEN
	HR.mCbBackward := TRUE;
ELSE
	HR.mCbBackward := FALSE;
	fin := TRUE;
END_IF
                    
END_ACTION

ACTION Store_W_active:
                      (*
Copyright (c) 2019 Manuel Goester, Michael Witt, Klaus Kammerer
Institute of Databases and Information Systems, Ulm University, Germany

Permission is hereby granted, free of charge, to any person obtaining a copy 
of this software and associated documentation files (the "Software"), to deal 
in the Software without restriction, including without limitation the rights 
to use, copy, modify, merge, publish, distribute, sublicense, and/or sell 
copies of the Software, and to permit persons to whom the Software is 
furnished to do so, subject to the following conditions:

The above copyright notice and this permission notice shall be included in 
all copies or substantial portions of the Software.

THE SOFTWARE IS PROVIDED "AS IS", WITHOUT WARRANTY OF ANY KIND, EXPRESS OR 
IMPLIED, INCLUDING BUT NOT LIMITED TO THE WARRANTIES OF MERCHANTABILITY, 
FITNESS FOR A PARTICULAR PURPOSE AND NONINFRINGEMENT. IN NO EVENT SHALL THE 
AUTHORS OR COPYRIGHT HOLDERS BE LIABLE FOR ANY CLAIM, DAMAGES OR OTHER 
LIABILITY, WHETHER IN AN ACTION OF CONTRACT, TORT OR OTHERWISE, ARISING FROM, 
OUT OF OR IN CONNECTION WITH THE SOFTWARE OR THE USE OR OTHER DEALINGS 
IN THE SOFTWARE.
*)
IF NOT hr_store_w.fin THEN
	hr_store_w(w:=TC.batchJobQueue.batchJobs[TC.currBatchJobIdx].workpieces[TC.batchJobQueue.batchJobs[TC.currBatchJobIdx].nextNotProcessedIdx]);
ELSE
	HR_SINGLE_MODE.subBlockStart := FALSE;
	
	// set BatchJobQueue to next workpiece

	HR.state := HR_State.FINISHED_SINGLE_MODE;
END_IF
                    
END_ACTION

ACTION ToDefaultPos_HR_STORE_W_active_active:
                      (*
Copyright (c) 2019 Manuel Goester, Michael Witt, Klaus Kammerer
Institute of Databases and Information Systems, Ulm University, Germany

Permission is hereby granted, free of charge, to any person obtaining a copy 
of this software and associated documentation files (the "Software"), to deal 
in the Software without restriction, including without limitation the rights 
to use, copy, modify, merge, publish, distribute, sublicense, and/or sell 
copies of the Software, and to permit persons to whom the Software is 
furnished to do so, subject to the following conditions:

The above copyright notice and this permission notice shall be included in 
all copies or substantial portions of the Software.

THE SOFTWARE IS PROVIDED "AS IS", WITHOUT WARRANTY OF ANY KIND, EXPRESS OR 
IMPLIED, INCLUDING BUT NOT LIMITED TO THE WARRANTIES OF MERCHANTABILITY, 
FITNESS FOR A PARTICULAR PURPOSE AND NONINFRINGEMENT. IN NO EVENT SHALL THE 
AUTHORS OR COPYRIGHT HOLDERS BE LIABLE FOR ANY CLAIM, DAMAGES OR OTHER 
LIABILITY, WHETHER IN AN ACTION OF CONTRACT, TORT OR OTHERWISE, ARISING FROM, 
OUT OF OR IN CONNECTION WITH THE SOFTWARE OR THE USE OR OTHER DEALINGS 
IN THE SOFTWARE.
*)
// returns the high rack TOWER to its default start position
// set "ausleger" arm to default position
IF HR.sCBack = FALSE THEN
	HR.mCBackward := TRUE;
ELSE 
	HR.mCBackward := FALSE;
	// set tower vertical position to max UP as well as horizontal position max RIGHT
	IF HR.sHorizontal = FALSE THEN
		HR.mHorizontalRight := TRUE;
	ELSE
		HR.mHorizontalRight := FALSE;
	END_IF
	
	IF HR.sVertical = FALSE THEN
		HR.mVerticalUp := TRUE;
	ELSE
		HR.mVerticalUp := FALSE;
	END_IF
END_IF
                    
END_ACTION

ACTION HR_WAIT_FOR_TC_active:
                      
                    
END_ACTION

ACTION HR_CONVEYOR_BACKWARD_exit:
                      (*
Copyright (c) 2019 Manuel Goester, Michael Witt, Klaus Kammerer
Institute of Databases and Information Systems, Ulm University, Germany

Permission is hereby granted, free of charge, to any person obtaining a copy 
of this software and associated documentation files (the "Software"), to deal 
in the Software without restriction, including without limitation the rights 
to use, copy, modify, merge, publish, distribute, sublicense, and/or sell 
copies of the Software, and to permit persons to whom the Software is 
furnished to do so, subject to the following conditions:

The above copyright notice and this permission notice shall be included in 
all copies or substantial portions of the Software.

THE SOFTWARE IS PROVIDED "AS IS", WITHOUT WARRANTY OF ANY KIND, EXPRESS OR 
IMPLIED, INCLUDING BUT NOT LIMITED TO THE WARRANTIES OF MERCHANTABILITY, 
FITNESS FOR A PARTICULAR PURPOSE AND NONINFRINGEMENT. IN NO EVENT SHALL THE 
AUTHORS OR COPYRIGHT HOLDERS BE LIABLE FOR ANY CLAIM, DAMAGES OR OTHER 
LIABILITY, WHETHER IN AN ACTION OF CONTRACT, TORT OR OTHERWISE, ARISING FROM, 
OUT OF OR IN CONNECTION WITH THE SOFTWARE OR THE USE OR OTHER DEALINGS 
IN THE SOFTWARE.
*)
fin := FALSE;
                    
END_ACTION

ACTION Init_active:
                      (*
Copyright (c) 2019 Manuel Goester, Michael Witt, Klaus Kammerer
Institute of Databases and Information Systems, Ulm University, Germany

Permission is hereby granted, free of charge, to any person obtaining a copy 
of this software and associated documentation files (the "Software"), to deal 
in the Software without restriction, including without limitation the rights 
to use, copy, modify, merge, publish, distribute, sublicense, and/or sell 
copies of the Software, and to permit persons to whom the Software is 
furnished to do so, subject to the following conditions:

The above copyright notice and this permission notice shall be included in 
all copies or substantial portions of the Software.

THE SOFTWARE IS PROVIDED "AS IS", WITHOUT WARRANTY OF ANY KIND, EXPRESS OR 
IMPLIED, INCLUDING BUT NOT LIMITED TO THE WARRANTIES OF MERCHANTABILITY, 
FITNESS FOR A PARTICULAR PURPOSE AND NONINFRINGEMENT. IN NO EVENT SHALL THE 
AUTHORS OR COPYRIGHT HOLDERS BE LIABLE FOR ANY CLAIM, DAMAGES OR OTHER 
LIABILITY, WHETHER IN AN ACTION OF CONTRACT, TORT OR OTHERWISE, ARISING FROM, 
OUT OF OR IN CONNECTION WITH THE SOFTWARE OR THE USE OR OTHER DEALINGS 
IN THE SOFTWARE.
*)
selectionValid := FALSE;
xFin := FALSE;
yFin := FALSE;
zFin := FALSE;
conveyorBeltFin := FALSE;
subBlockStart := FALSE;
calibrateYAxis := 0;
step := 1;
                    
END_ACTION

ACTION ConveyorBack_HR_STORE_W_active_entry:
                      (*
Copyright (c) 2019 Manuel Goester, Michael Witt, Klaus Kammerer
Institute of Databases and Information Systems, Ulm University, Germany

Permission is hereby granted, free of charge, to any person obtaining a copy 
of this software and associated documentation files (the "Software"), to deal 
in the Software without restriction, including without limitation the rights 
to use, copy, modify, merge, publish, distribute, sublicense, and/or sell 
copies of the Software, and to permit persons to whom the Software is 
furnished to do so, subject to the following conditions:

The above copyright notice and this permission notice shall be included in 
all copies or substantial portions of the Software.

THE SOFTWARE IS PROVIDED "AS IS", WITHOUT WARRANTY OF ANY KIND, EXPRESS OR 
IMPLIED, INCLUDING BUT NOT LIMITED TO THE WARRANTIES OF MERCHANTABILITY, 
FITNESS FOR A PARTICULAR PURPOSE AND NONINFRINGEMENT. IN NO EVENT SHALL THE 
AUTHORS OR COPYRIGHT HOLDERS BE LIABLE FOR ANY CLAIM, DAMAGES OR OTHER 
LIABILITY, WHETHER IN AN ACTION OF CONTRACT, TORT OR OTHERWISE, ARISING FROM, 
OUT OF OR IN CONNECTION WITH THE SOFTWARE OR THE USE OR OTHER DEALINGS 
IN THE SOFTWARE.
*)
SM.currW.linePos := 0;
HR.state := HR_State.STORE_W;
                    
END_ACTION

ACTION HR_CALIBRATE_Y_AXIS_active:
                      (*
Copyright (c) 2019 Manuel Goester, Michael Witt, Klaus Kammerer
Institute of Databases and Information Systems, Ulm University, Germany

Permission is hereby granted, free of charge, to any person obtaining a copy 
of this software and associated documentation files (the "Software"), to deal 
in the Software without restriction, including without limitation the rights 
to use, copy, modify, merge, publish, distribute, sublicense, and/or sell 
copies of the Software, and to permit persons to whom the Software is 
furnished to do so, subject to the following conditions:

The above copyright notice and this permission notice shall be included in 
all copies or substantial portions of the Software.

THE SOFTWARE IS PROVIDED "AS IS", WITHOUT WARRANTY OF ANY KIND, EXPRESS OR 
IMPLIED, INCLUDING BUT NOT LIMITED TO THE WARRANTIES OF MERCHANTABILITY, 
FITNESS FOR A PARTICULAR PURPOSE AND NONINFRINGEMENT. IN NO EVENT SHALL THE 
AUTHORS OR COPYRIGHT HOLDERS BE LIABLE FOR ANY CLAIM, DAMAGES OR OTHER 
LIABILITY, WHETHER IN AN ACTION OF CONTRACT, TORT OR OTHERWISE, ARISING FROM, 
OUT OF OR IN CONNECTION WITH THE SOFTWARE OR THE USE OR OTHER DEALINGS 
IN THE SOFTWARE.
*)
IF calibrateYAxis = 2 THEN
	IF NOT(HR.sVertical) THEN
		HR.mVerticalUp := TRUE;
	ELSE
		Hr.mVerticalUp := FALSE;
		Hr.cY := 0;
		fin := TRUE;
		calibrateYAxis := 0;
	END_IF
ELSE
	IF NOT(alreadyCounted) THEN
		calibrateYAxis := calibrateYAxis + 1;
		alreadyCounted := TRUE;
	ELSE
		fin := TRUE;
	END_IF
END_IF
                    
END_ACTION

ACTION HR_CALIBRATE_Y_AXIS_exit:
                      (*
Copyright (c) 2019 Manuel Goester, Michael Witt, Klaus Kammerer
Institute of Databases and Information Systems, Ulm University, Germany

Permission is hereby granted, free of charge, to any person obtaining a copy 
of this software and associated documentation files (the "Software"), to deal 
in the Software without restriction, including without limitation the rights 
to use, copy, modify, merge, publish, distribute, sublicense, and/or sell 
copies of the Software, and to permit persons to whom the Software is 
furnished to do so, subject to the following conditions:

The above copyright notice and this permission notice shall be included in 
all copies or substantial portions of the Software.

THE SOFTWARE IS PROVIDED "AS IS", WITHOUT WARRANTY OF ANY KIND, EXPRESS OR 
IMPLIED, INCLUDING BUT NOT LIMITED TO THE WARRANTIES OF MERCHANTABILITY, 
FITNESS FOR A PARTICULAR PURPOSE AND NONINFRINGEMENT. IN NO EVENT SHALL THE 
AUTHORS OR COPYRIGHT HOLDERS BE LIABLE FOR ANY CLAIM, DAMAGES OR OTHER 
LIABILITY, WHETHER IN AN ACTION OF CONTRACT, TORT OR OTHERWISE, ARISING FROM, 
OUT OF OR IN CONNECTION WITH THE SOFTWARE OR THE USE OR OTHER DEALINGS 
IN THE SOFTWARE.
*)
fin := FALSE;
alreadyCounted := FALSE;
                    
END_ACTION

ACTION HR_CONVEYOR_FORWARD_exit:
                      (*
Copyright (c) 2019 Manuel Goester, Michael Witt, Klaus Kammerer
Institute of Databases and Information Systems, Ulm University, Germany

Permission is hereby granted, free of charge, to any person obtaining a copy 
of this software and associated documentation files (the "Software"), to deal 
in the Software without restriction, including without limitation the rights 
to use, copy, modify, merge, publish, distribute, sublicense, and/or sell 
copies of the Software, and to permit persons to whom the Software is 
furnished to do so, subject to the following conditions:

The above copyright notice and this permission notice shall be included in 
all copies or substantial portions of the Software.

THE SOFTWARE IS PROVIDED "AS IS", WITHOUT WARRANTY OF ANY KIND, EXPRESS OR 
IMPLIED, INCLUDING BUT NOT LIMITED TO THE WARRANTIES OF MERCHANTABILITY, 
FITNESS FOR A PARTICULAR PURPOSE AND NONINFRINGEMENT. IN NO EVENT SHALL THE 
AUTHORS OR COPYRIGHT HOLDERS BE LIABLE FOR ANY CLAIM, DAMAGES OR OTHER 
LIABILITY, WHETHER IN AN ACTION OF CONTRACT, TORT OR OTHERWISE, ARISING FROM, 
OUT OF OR IN CONNECTION WITH THE SOFTWARE OR THE USE OR OTHER DEALINGS 
IN THE SOFTWARE.
*)
fin := FALSE;
                    
END_ACTION

ACTION HR_CONVEYOR_FORWARD_active:
                      (*
Copyright (c) 2019 Manuel Goester, Michael Witt, Klaus Kammerer
Institute of Databases and Information Systems, Ulm University, Germany

Permission is hereby granted, free of charge, to any person obtaining a copy 
of this software and associated documentation files (the "Software"), to deal 
in the Software without restriction, including without limitation the rights 
to use, copy, modify, merge, publish, distribute, sublicense, and/or sell 
copies of the Software, and to permit persons to whom the Software is 
furnished to do so, subject to the following conditions:

The above copyright notice and this permission notice shall be included in 
all copies or substantial portions of the Software.

THE SOFTWARE IS PROVIDED "AS IS", WITHOUT WARRANTY OF ANY KIND, EXPRESS OR 
IMPLIED, INCLUDING BUT NOT LIMITED TO THE WARRANTIES OF MERCHANTABILITY, 
FITNESS FOR A PARTICULAR PURPOSE AND NONINFRINGEMENT. IN NO EVENT SHALL THE 
AUTHORS OR COPYRIGHT HOLDERS BE LIABLE FOR ANY CLAIM, DAMAGES OR OTHER 
LIABILITY, WHETHER IN AN ACTION OF CONTRACT, TORT OR OTHERWISE, ARISING FROM, 
OUT OF OR IN CONNECTION WITH THE SOFTWARE OR THE USE OR OTHER DEALINGS 
IN THE SOFTWARE.
*)
IF HR.lbOut THEN
	HR.mCbForward := TRUE;
ELSE
	HR.mCbForward := FALSE;
	fin := TRUE; 
END_IF
                    
END_ACTION

ACTION HR_STORES_W_exit:
                      (*
Copyright (c) 2019 Manuel Goester, Michael Witt, Klaus Kammerer
Institute of Databases and Information Systems, Ulm University, Germany

Permission is hereby granted, free of charge, to any person obtaining a copy 
of this software and associated documentation files (the "Software"), to deal 
in the Software without restriction, including without limitation the rights 
to use, copy, modify, merge, publish, distribute, sublicense, and/or sell 
copies of the Software, and to permit persons to whom the Software is 
furnished to do so, subject to the following conditions:

The above copyright notice and this permission notice shall be included in 
all copies or substantial portions of the Software.

THE SOFTWARE IS PROVIDED "AS IS", WITHOUT WARRANTY OF ANY KIND, EXPRESS OR 
IMPLIED, INCLUDING BUT NOT LIMITED TO THE WARRANTIES OF MERCHANTABILITY, 
FITNESS FOR A PARTICULAR PURPOSE AND NONINFRINGEMENT. IN NO EVENT SHALL THE 
AUTHORS OR COPYRIGHT HOLDERS BE LIABLE FOR ANY CLAIM, DAMAGES OR OTHER 
LIABILITY, WHETHER IN AN ACTION OF CONTRACT, TORT OR OTHERWISE, ARISING FROM, 
OUT OF OR IN CONNECTION WITH THE SOFTWARE OR THE USE OR OTHER DEALINGS 
IN THE SOFTWARE.
*)
fin := FALSE;
                    
END_ACTION

ACTION HR_SET_TC_STATE_exit:
                      (*
Copyright (c) 2019 Manuel Goester, Michael Witt, Klaus Kammerer
Institute of Databases and Information Systems, Ulm University, Germany

Permission is hereby granted, free of charge, to any person obtaining a copy 
of this software and associated documentation files (the "Software"), to deal 
in the Software without restriction, including without limitation the rights 
to use, copy, modify, merge, publish, distribute, sublicense, and/or sell 
copies of the Software, and to permit persons to whom the Software is 
furnished to do so, subject to the following conditions:

The above copyright notice and this permission notice shall be included in 
all copies or substantial portions of the Software.

THE SOFTWARE IS PROVIDED "AS IS", WITHOUT WARRANTY OF ANY KIND, EXPRESS OR 
IMPLIED, INCLUDING BUT NOT LIMITED TO THE WARRANTIES OF MERCHANTABILITY, 
FITNESS FOR A PARTICULAR PURPOSE AND NONINFRINGEMENT. IN NO EVENT SHALL THE 
AUTHORS OR COPYRIGHT HOLDERS BE LIABLE FOR ANY CLAIM, DAMAGES OR OTHER 
LIABILITY, WHETHER IN AN ACTION OF CONTRACT, TORT OR OTHERWISE, ARISING FROM, 
OUT OF OR IN CONNECTION WITH THE SOFTWARE OR THE USE OR OTHER DEALINGS 
IN THE SOFTWARE.
*)
fin := FALSE;
                    
END_ACTION

ACTION HR_SET_TC_STATE_active:
                      (*
Copyright (c) 2019 Manuel Goester, Michael Witt, Klaus Kammerer
Institute of Databases and Information Systems, Ulm University, Germany

Permission is hereby granted, free of charge, to any person obtaining a copy 
of this software and associated documentation files (the "Software"), to deal 
in the Software without restriction, including without limitation the rights 
to use, copy, modify, merge, publish, distribute, sublicense, and/or sell 
copies of the Software, and to permit persons to whom the Software is 
furnished to do so, subject to the following conditions:

The above copyright notice and this permission notice shall be included in 
all copies or substantial portions of the Software.

THE SOFTWARE IS PROVIDED "AS IS", WITHOUT WARRANTY OF ANY KIND, EXPRESS OR 
IMPLIED, INCLUDING BUT NOT LIMITED TO THE WARRANTIES OF MERCHANTABILITY, 
FITNESS FOR A PARTICULAR PURPOSE AND NONINFRINGEMENT. IN NO EVENT SHALL THE 
AUTHORS OR COPYRIGHT HOLDERS BE LIABLE FOR ANY CLAIM, DAMAGES OR OTHER 
LIABILITY, WHETHER IN AN ACTION OF CONTRACT, TORT OR OTHERWISE, ARISING FROM, 
OUT OF OR IN CONNECTION WITH THE SOFTWARE OR THE USE OR OTHER DEALINGS 
IN THE SOFTWARE.
*)
IF NOT(fin) THEN
	IF TC.state = TC_State.W_LOADED THEN
		// workpiece was already loaded by a multi mode batchjob which has been running before this batch job
		// so dont load a now one
		// OR
		// the batch job before was a single mode batch job. So this batch job loaded its workpiece itself
		// now it is loaded, so production can start
		// signalise that production starts
		TC.state := TC_State.WAIT_UNTIL_W_FINISHED;
		fin := TRUE;
	ELSE
		// load a new workpiece
		TC.state := TC_State.LOAD_NEXT_W;
	END_IF
END_IF

                    
END_ACTION
END_PROGRAM

PROGRAM MAIN
  VAR
    workpieces : ARRAY[1..9] OF Workpiece;
    format : Format;
    format1 : Format;
    format2 : Format;
    format3 : Format;
    format4 : Format;
    format5 : Format;
    format6 : Format;
    format7 : Format;
    format8 : Format;
    format9 : Format;
    format10 : Format;
    format11 : Format;
    format12 : Format;
    format13 : Format;
    format14 : Format;
    format15 : Format;
    format16 : Format;
    newWorkpi : Workpiece;
  END_VAR

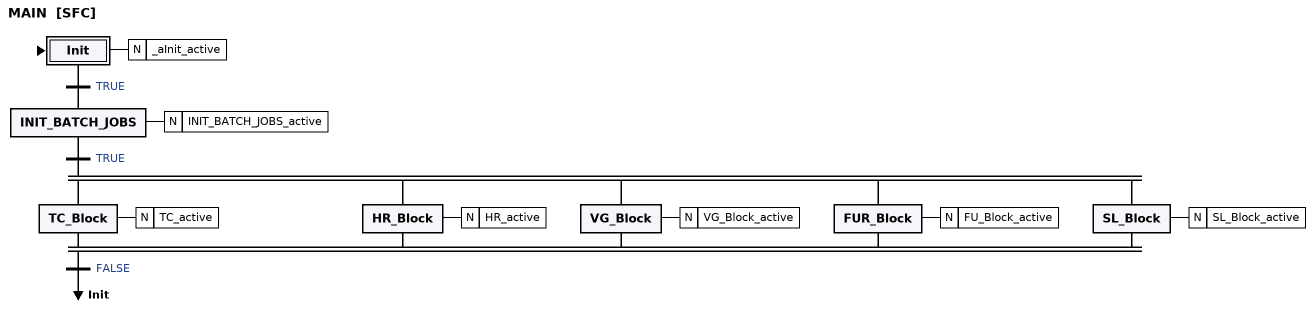
INITIAL_STEP Init:
  _aInit_active(N);
END_STEP
TRANSITION FROM Init TO INIT_BATCH_JOBS
  := TRUE;
END_TRANSITION
STEP INIT_BATCH_JOBS:
  INIT_BATCH_JOBS_active(N);
END_STEP
TRANSITION FROM INIT_BATCH_JOBS TO (TC_Block, HR_Block, VG_Block, FUR_Block, SL_Block)
  := TRUE;
END_TRANSITION
STEP TC_Block:
  TC_active(N);
END_STEP
TRANSITION FROM (TC_Block, HR_Block, VG_Block, FUR_Block, SL_Block) TO Init
  := FALSE;
END_TRANSITION
STEP HR_Block:
  HR_active(N);
END_STEP
STEP VG_Block:
  VG_Block_active(N);
END_STEP
STEP FUR_Block:
  FU_Block_active(N);
END_STEP
STEP SL_Block:
  SL_Block_active(N);
END_STEP

ACTION FU_Block_active:
                      (*
Copyright (c) 2019 Manuel Goester, Michael Witt, Klaus Kammerer
Institute of Databases and Information Systems, Ulm University, Germany

Permission is hereby granted, free of charge, to any person obtaining a copy 
of this software and associated documentation files (the "Software"), to deal 
in the Software without restriction, including without limitation the rights 
to use, copy, modify, merge, publish, distribute, sublicense, and/or sell 
copies of the Software, and to permit persons to whom the Software is 
furnished to do so, subject to the following conditions:

The above copyright notice and this permission notice shall be included in 
all copies or substantial portions of the Software.

THE SOFTWARE IS PROVIDED "AS IS", WITHOUT WARRANTY OF ANY KIND, EXPRESS OR 
IMPLIED, INCLUDING BUT NOT LIMITED TO THE WARRANTIES OF MERCHANTABILITY, 
FITNESS FOR A PARTICULAR PURPOSE AND NONINFRINGEMENT. IN NO EVENT SHALL THE 
AUTHORS OR COPYRIGHT HOLDERS BE LIABLE FOR ANY CLAIM, DAMAGES OR OTHER 
LIABILITY, WHETHER IN AN ACTION OF CONTRACT, TORT OR OTHERWISE, ARISING FROM, 
OUT OF OR IN CONNECTION WITH THE SOFTWARE OR THE USE OR OTHER DEALINGS 
IN THE SOFTWARE.
*)
FUR.any_motor_running := FUR.compressor AND FUR.mRaClockwise AND FUR.mRaCClockwise AND FUR.mConveyorBeltForward AND FUR.mSaw AND FUR.mFurnanceSliderIn  AND FUR.mFurnanceSliderOut AND FUR.mSuckertoFurnance AND FUR.mSuckertoRa AND FUR.compressor  AND FUR.valveVacuum AND FUR.valveLowering AND FUR.valveFurnanceDoor AND FUR.valveSlider;

IF (TC_POU.started OR FUR.any_motor_running) AND NOT(TC.instant_shutdown) THEN
	IF TC.mode_active = ExecutionMode.single THEN
		FUR_SINGLE_MODE();
	ELSIF TC.mode_active = ExecutionMode.multi THEN
		FUR_MULTI_MODE();
	END_IF
ELSE
	// instant shutdown --> all motors off
	FUR.compressor 				:= FALSE;
	FUR.mRaClockwise 			:= FALSE;
	FUR.mRaCClockwise  			:= FALSE;
	FUR.mConveyorBeltForward	:= FALSE;
	FUR.mSaw  					:= FALSE;
	FUR.mFurnanceSliderIn 		:= FALSE;
	FUR.mFurnanceSliderOut 		:= FALSE;
	FUR.mSuckertoFurnance 		:= FALSE;
	FUR.mSuckertoRa 			:= FALSE;
	FUR.compressor 				:= FALSE;
	FUR.valveVacuum				:= FALSE;
	FUR.valveLowering			:= FALSE;
	FUR.valveFurnanceDoor		:= FALSE;
	FUR.valveSlider 			:= FALSE;
END_IF
                    
END_ACTION

ACTION VG_Block_active:
                      (*
Copyright (c) 2019 Manuel Goester, Michael Witt, Klaus Kammerer
Institute of Databases and Information Systems, Ulm University, Germany

Permission is hereby granted, free of charge, to any person obtaining a copy 
of this software and associated documentation files (the "Software"), to deal 
in the Software without restriction, including without limitation the rights 
to use, copy, modify, merge, publish, distribute, sublicense, and/or sell 
copies of the Software, and to permit persons to whom the Software is 
furnished to do so, subject to the following conditions:

The above copyright notice and this permission notice shall be included in 
all copies or substantial portions of the Software.

THE SOFTWARE IS PROVIDED "AS IS", WITHOUT WARRANTY OF ANY KIND, EXPRESS OR 
IMPLIED, INCLUDING BUT NOT LIMITED TO THE WARRANTIES OF MERCHANTABILITY, 
FITNESS FOR A PARTICULAR PURPOSE AND NONINFRINGEMENT. IN NO EVENT SHALL THE 
AUTHORS OR COPYRIGHT HOLDERS BE LIABLE FOR ANY CLAIM, DAMAGES OR OTHER 
LIABILITY, WHETHER IN AN ACTION OF CONTRACT, TORT OR OTHERWISE, ARISING FROM, 
OUT OF OR IN CONNECTION WITH THE SOFTWARE OR THE USE OR OTHER DEALINGS 
IN THE SOFTWARE.
*)
VG.any_motor_running := VG.mHorizontalBackward OR VG.mHorizontalForward OR VG.mRotationCClockwise OR VG.mRotationClockwise OR VG.mVerticalDown OR VG.mVerticalUp;

IF (TC_POU.started OR VG.any_motor_running) AND NOT(TC.instant_shutdown) THEN
	IF TC.mode_active = ExecutionMode.single THEN
		VG_SINGLE_MODE();
	ELSIF TC.mode_active = ExecutionMode.multi THEN
		VG_MULTI_MODE();
	END_IF
ELSE
	// instant shutdown --> all motors off
	VG.mHorizontalBackward 	:= FALSE;
	VG.mHorizontalForward 	:= FALSE;
	VG.mRotationCClockwise 	:= FALSE;
	VG.mRotationClockwise 	:= FALSE;
	VG.mVerticalDown 		:= FALSE; 
	VG.mVerticalUp 			:= FALSE;
END_IF
                    
END_ACTION

ACTION SL_Block_active:
                      (*
Copyright (c) 2019 Manuel Goester, Michael Witt, Klaus Kammerer
Institute of Databases and Information Systems, Ulm University, Germany

Permission is hereby granted, free of charge, to any person obtaining a copy 
of this software and associated documentation files (the "Software"), to deal 
in the Software without restriction, including without limitation the rights 
to use, copy, modify, merge, publish, distribute, sublicense, and/or sell 
copies of the Software, and to permit persons to whom the Software is 
furnished to do so, subject to the following conditions:

The above copyright notice and this permission notice shall be included in 
all copies or substantial portions of the Software.

THE SOFTWARE IS PROVIDED "AS IS", WITHOUT WARRANTY OF ANY KIND, EXPRESS OR 
IMPLIED, INCLUDING BUT NOT LIMITED TO THE WARRANTIES OF MERCHANTABILITY, 
FITNESS FOR A PARTICULAR PURPOSE AND NONINFRINGEMENT. IN NO EVENT SHALL THE 
AUTHORS OR COPYRIGHT HOLDERS BE LIABLE FOR ANY CLAIM, DAMAGES OR OTHER 
LIABILITY, WHETHER IN AN ACTION OF CONTRACT, TORT OR OTHERWISE, ARISING FROM, 
OUT OF OR IN CONNECTION WITH THE SOFTWARE OR THE USE OR OTHER DEALINGS 
IN THE SOFTWARE.
*)
SL.any_motor_running := SL.mConveyorBelt AND SL.compressor;

IF (TC_POU.started OR SL.any_motor_running) AND NOT(TC.instant_shutdown) THEN
	IF TC.mode_active = ExecutionMode.single THEN
		SL_SINGLE_MODE();
	ELSIF TC.mode_active = ExecutionMode.multi THEN
		SL_MULTI_MODE();
	END_IF
ELSE
	// instant shutdown --> all motors off
	SL.mConveyorBelt 	:= FALSE;
	SL.compressor		:= FALSE;
END_IF
                    
END_ACTION

ACTION TC_active:
                      (*
Copyright (c) 2019 Manuel Goester, Michael Witt, Klaus Kammerer
Institute of Databases and Information Systems, Ulm University, Germany

Permission is hereby granted, free of charge, to any person obtaining a copy 
of this software and associated documentation files (the "Software"), to deal 
in the Software without restriction, including without limitation the rights 
to use, copy, modify, merge, publish, distribute, sublicense, and/or sell 
copies of the Software, and to permit persons to whom the Software is 
furnished to do so, subject to the following conditions:

The above copyright notice and this permission notice shall be included in 
all copies or substantial portions of the Software.

THE SOFTWARE IS PROVIDED "AS IS", WITHOUT WARRANTY OF ANY KIND, EXPRESS OR 
IMPLIED, INCLUDING BUT NOT LIMITED TO THE WARRANTIES OF MERCHANTABILITY, 
FITNESS FOR A PARTICULAR PURPOSE AND NONINFRINGEMENT. IN NO EVENT SHALL THE 
AUTHORS OR COPYRIGHT HOLDERS BE LIABLE FOR ANY CLAIM, DAMAGES OR OTHER 
LIABILITY, WHETHER IN AN ACTION OF CONTRACT, TORT OR OTHERWISE, ARISING FROM, 
OUT OF OR IN CONNECTION WITH THE SOFTWARE OR THE USE OR OTHER DEALINGS 
IN THE SOFTWARE.
*)
// invoke TC_POU program
TC_POU();
                    
END_ACTION

ACTION HR_active:
                      (*
Copyright (c) 2019 Manuel Goester, Michael Witt, Klaus Kammerer
Institute of Databases and Information Systems, Ulm University, Germany

Permission is hereby granted, free of charge, to any person obtaining a copy 
of this software and associated documentation files (the "Software"), to deal 
in the Software without restriction, including without limitation the rights 
to use, copy, modify, merge, publish, distribute, sublicense, and/or sell 
copies of the Software, and to permit persons to whom the Software is 
furnished to do so, subject to the following conditions:

The above copyright notice and this permission notice shall be included in 
all copies or substantial portions of the Software.

THE SOFTWARE IS PROVIDED "AS IS", WITHOUT WARRANTY OF ANY KIND, EXPRESS OR 
IMPLIED, INCLUDING BUT NOT LIMITED TO THE WARRANTIES OF MERCHANTABILITY, 
FITNESS FOR A PARTICULAR PURPOSE AND NONINFRINGEMENT. IN NO EVENT SHALL THE 
AUTHORS OR COPYRIGHT HOLDERS BE LIABLE FOR ANY CLAIM, DAMAGES OR OTHER 
LIABILITY, WHETHER IN AN ACTION OF CONTRACT, TORT OR OTHERWISE, ARISING FROM, 
OUT OF OR IN CONNECTION WITH THE SOFTWARE OR THE USE OR OTHER DEALINGS 
IN THE SOFTWARE.
*)
HR.any_motor_running := HR.mCBackward OR HR.mCForward OR HR.mCbBackward OR HR.mCbForward OR HR.mHorizontalLeft OR HR.mHorizontalRight OR HR.mVerticalDown OR HR.mVerticalUp;
// invoke the appropriate HR program that fits to the execution mode of the current batch job
IF (TC.batchJobQueue.batchJobs[TC.currBatchJobIdx].state = BatchJobState.STARTED OR HR.any_motor_running) AND NOT(TC.instant_shutdown) THEN
	IF TC.mode_active = ExecutionMode.single THEN
		HR_SINGLE_MODE();
	ELSIF TC.mode_active = ExecutionMode.multi THEN
		HR_MULTI_MODE();
	ELSIF TC.mode_active = ExecutionMode.sorting THEN
		HR.state := HR_State.SORTING;
		HR_SORTING_MODE();
	END_IF
ELSE
	// instant shutdown --> all motors off
	HR.mCBackward 		:= FALSE;
	HR.mCForward  		:= FALSE;
	HR.mCbBackward 		:= FALSE;
	HR.mCbForward  		:= FALSE;
	HR.mHorizontalLeft 	:= FALSE;
	HR.mHorizontalRight := FALSE;
	HR.mVerticalDown 	:= FALSE;
	HR.mVerticalUp 		:= FALSE;
END_IF
                    
END_ACTION

ACTION _aInit_active:
                      (*
Copyright (c) 2019 Manuel Goester, Michael Witt, Klaus Kammerer
Institute of Databases and Information Systems, Ulm University, Germany

Permission is hereby granted, free of charge, to any person obtaining a copy 
of this software and associated documentation files (the "Software"), to deal 
in the Software without restriction, including without limitation the rights 
to use, copy, modify, merge, publish, distribute, sublicense, and/or sell 
copies of the Software, and to permit persons to whom the Software is 
furnished to do so, subject to the following conditions:

The above copyright notice and this permission notice shall be included in 
all copies or substantial portions of the Software.

THE SOFTWARE IS PROVIDED "AS IS", WITHOUT WARRANTY OF ANY KIND, EXPRESS OR 
IMPLIED, INCLUDING BUT NOT LIMITED TO THE WARRANTIES OF MERCHANTABILITY, 
FITNESS FOR A PARTICULAR PURPOSE AND NONINFRINGEMENT. IN NO EVENT SHALL THE 
AUTHORS OR COPYRIGHT HOLDERS BE LIABLE FOR ANY CLAIM, DAMAGES OR OTHER 
LIABILITY, WHETHER IN AN ACTION OF CONTRACT, TORT OR OTHERWISE, ARISING FROM, 
OUT OF OR IN CONNECTION WITH THE SOFTWARE OR THE USE OR OTHER DEALINGS 
IN THE SOFTWARE.
*)
// program has been started
TC.is_plc_running := TRUE;

// init some vars
TC.currBatchJobIdx := 1;
HR.any_motor_running := HR.mCBackward OR HR.mCForward OR HR.mCbBackward OR HR.mCbForward OR HR.mHorizontalLeft OR HR.mHorizontalRight OR HR.mVerticalDown OR HR.mVerticalUp;
VG.any_motor_running := VG.mHorizontalBackward OR VG.mHorizontalForward OR VG.mRotationCClockwise OR VG.mRotationClockwise OR VG.mVerticalDown OR VG.mVerticalUp;
FUR.any_motor_running := FUR.compressor AND FUR.mRaClockwise AND FUR.mRaCClockwise AND FUR.mConveyorBeltForward AND FUR.mSaw AND FUR.mFurnanceSliderIn  AND FUR.mFurnanceSliderOut AND FUR.mSuckertoFurnance AND FUR.mSuckertoRa AND FUR.compressor  AND FUR.valveVacuum AND FUR.valveLowering AND FUR.valveFurnanceDoor AND FUR.valveSlider;
SL.any_motor_running := SL.mConveyorBelt AND SL.compressor;
                    
END_ACTION

ACTION INIT_BATCH_JOBS_active:
                      (*
	BatchJobs, which shall run on the DBIS Factory, will be initialized here
	By using the funciton TC_FUNs/addBatchJobToQueue a BatchJob can be added to the queue, e.g. by calling it via UA server

Copyright (c) 2019 Manuel Goester, Michael Witt, Klaus Kammerer
Institute of Databases and Information Systems, Ulm University, Germany

Permission is hereby granted, free of charge, to any person obtaining a copy 
of this software and associated documentation files (the "Software"), to deal 
in the Software without restriction, including without limitation the rights 
to use, copy, modify, merge, publish, distribute, sublicense, and/or sell 
copies of the Software, and to permit persons to whom the Software is 
furnished to do so, subject to the following conditions:

The above copyright notice and this permission notice shall be included in 
all copies or substantial portions of the Software.

THE SOFTWARE IS PROVIDED "AS IS", WITHOUT WARRANTY OF ANY KIND, EXPRESS OR 
IMPLIED, INCLUDING BUT NOT LIMITED TO THE WARRANTIES OF MERCHANTABILITY, 
FITNESS FOR A PARTICULAR PURPOSE AND NONINFRINGEMENT. IN NO EVENT SHALL THE 
AUTHORS OR COPYRIGHT HOLDERS BE LIABLE FOR ANY CLAIM, DAMAGES OR OTHER 
LIABILITY, WHETHER IN AN ACTION OF CONTRACT, TORT OR OTHERWISE, ARISING FROM, 
OUT OF OR IN CONNECTION WITH THE SOFTWARE OR THE USE OR OTHER DEALINGS 
IN THE SOFTWARE.
*)

(*
	Defining formats
*)
format1 := newFormat(FALSE, FALSE, FALSE, FALSE, T#5S, T#5S);
format2 := newFormat(FALSE, FALSE, FALSE, TRUE,  T#5S, T#5S);
format3 := newFormat(FALSE, FALSE, TRUE,  FALSE, T#5S, T#5S);
format4 := newFormat(FALSE, FALSE, TRUE,  TRUE,  T#5S, T#5S);

format5 := newFormat(FALSE, TRUE, FALSE, FALSE, T#5S, T#5S);
format6 := newFormat(FALSE, TRUE, FALSE, TRUE,  T#5S, T#5S);
format7 := newFormat(FALSE, TRUE, TRUE,  FALSE, T#5S, T#5S);
format8 := newFormat(FALSE, TRUE, TRUE,  TRUE,  T#5S, T#5S);

format9 := newFormat(TRUE, FALSE, FALSE, FALSE, T#5S, T#5S);
format10:= newFormat(TRUE, FALSE, FALSE, TRUE,  T#5S, T#5S);
format11:= newFormat(TRUE, FALSE, TRUE,  FALSE, T#5S, T#5S);
format12:= newFormat(TRUE, FALSE, TRUE,  TRUE,  T#5S, T#5S);

format13:= newFormat(TRUE, TRUE, FALSE, FALSE, T#5S, T#5S);
format14:= newFormat(TRUE, TRUE, FALSE, TRUE,  T#5S, T#5S);
format15:= newFormat(TRUE, TRUE, TRUE,  FALSE, T#5S, T#5S);
format16:= newFormat(TRUE, TRUE, TRUE,  TRUE,  T#5S, T#5S);

(*
	Testcase 1: SINGLE MODE
*)

workpieces[1] := newWorkpiece('unknown', W_State.AT_RACK_22, RackPos.RACK_22, RackPos.RACK_22, format15);
workpieces[2] := newWorkpiece('unknown', W_State.AT_RACK_23, RackPos.RACK_23, RackPos.RACK_23, format16);
workpieces[3] := newWorkpiece('unknown', W_State.AT_RACK_13, RackPos.RACK_13, RackPos.RACK_13, format8);
workpieces[4] := newWorkpiece('unknown', W_State.AT_RACK_21, RackPos.RACK_21, RackPos.RACK_21, format16);
workpieces[5] := newWorkpiece('unknown', W_State.AT_RACK_11, RackPos.RACK_11, RackPos.RACK_11, format15);
workpieces[6] := newWorkpiece('unknown', W_State.AT_RACK_12, RackPos.RACK_12, RackPos.RACK_12, format15);
addBatchJobToQueue(newbatchJob(6, workpieces, ExecutionMode.single));



(*
	Testcase 2: MULTI MODE
*)
(*
workpieces[1] := newWorkpiece('unknown', W_State.AT_RACK_22, RackPos.RACK_22, RackPos.RACK_22, format15);
workpieces[2] := newWorkpiece('unknown', W_State.AT_RACK_23, RackPos.RACK_23, RackPos.RACK_23, format16);
workpieces[3] := newWorkpiece('unknown', W_State.AT_RACK_13, RackPos.RACK_13, RackPos.RACK_13, format8);
workpieces[4] := newWorkpiece('unknown', W_State.AT_RACK_21, RackPos.RACK_21, RackPos.RACK_21, format16);
workpieces[5] := newWorkpiece('unknown', W_State.AT_RACK_11, RackPos.RACK_11, RackPos.RACK_11, format15);
workpieces[6] := newWorkpiece('unknown', W_State.AT_RACK_12, RackPos.RACK_12, RackPos.RACK_12, format15);
addBatchJobToQueue(newbatchJob(6, workpieces, ExecutionMode.multi));
*)


(*
	Testcase 3: SORTING MODE
*)
(*
workpieces[1] := newWorkpiece('unknown', W_State.AT_RACK_22, RackPos.RACK_22, RackPos.RACK_22, format15);
workpieces[2] := newWorkpiece('unknown', W_State.AT_RACK_23, RackPos.RACK_23, RackPos.RACK_23, format16);
workpieces[3] := newWorkpiece('unknown', W_State.AT_RACK_13, RackPos.RACK_13, RackPos.RACK_13, format8);
workpieces[4] := newWorkpiece('unknown', W_State.AT_RACK_21, RackPos.RACK_21, RackPos.RACK_21, format16);
addBatchJobToQueue(newbatchJob(4, workpieces, ExecutionMode.sorting));
*)
                    
END_ACTION
END_PROGRAM

PROGRAM SL_MULTI_MODE
  VAR
    fin : BOOL;
    sl_fb : SL_FB;
    step : INT := 1;
  END_VAR

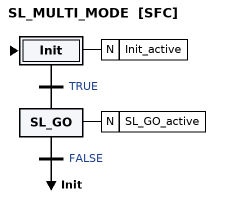
INITIAL_STEP Init:
  Init_active(N);
END_STEP
TRANSITION FROM Init TO SL_GO
  := TRUE;
END_TRANSITION
STEP SL_GO:
  SL_GO_active(N);
END_STEP
TRANSITION FROM SL_GO TO Init
  := FALSE;
END_TRANSITION

ACTION SL_GO_active:
                      (*
Copyright (c) 2019 Manuel Goester, Michael Witt, Klaus Kammerer
Institute of Databases and Information Systems, Ulm University, Germany

Permission is hereby granted, free of charge, to any person obtaining a copy 
of this software and associated documentation files (the "Software"), to deal 
in the Software without restriction, including without limitation the rights 
to use, copy, modify, merge, publish, distribute, sublicense, and/or sell 
copies of the Software, and to permit persons to whom the Software is 
furnished to do so, subject to the following conditions:

The above copyright notice and this permission notice shall be included in 
all copies or substantial portions of the Software.

THE SOFTWARE IS PROVIDED "AS IS", WITHOUT WARRANTY OF ANY KIND, EXPRESS OR 
IMPLIED, INCLUDING BUT NOT LIMITED TO THE WARRANTIES OF MERCHANTABILITY, 
FITNESS FOR A PARTICULAR PURPOSE AND NONINFRINGEMENT. IN NO EVENT SHALL THE 
AUTHORS OR COPYRIGHT HOLDERS BE LIABLE FOR ANY CLAIM, DAMAGES OR OTHER 
LIABILITY, WHETHER IN AN ACTION OF CONTRACT, TORT OR OTHERWISE, ARISING FROM, 
OUT OF OR IN CONNECTION WITH THE SOFTWARE OR THE USE OR OTHER DEALINGS 
IN THE SOFTWARE.
*)
CASE step OF
	1:
		IF SL.currW.state <> W_State.NULL AND SL.state = SL_State.WAITING_FOR_W THEN
			SL.state := SL_State.W_RECEIVED;
			step := step + 1;
		END_IF
	2:
		IF NOT(fin) THEN
			sl_fb();
			fin := sl_fb.fin;
		ELSE
			// wait for VG to pick up w
			SL.state := SL_State.WAITING_FOR_VG_TO_PICK_UP_W;
			step := step + 1;
		END_IF
	3:
		IF VG.state = VG_State.TO_SL_TAKE_W_FINISHED OR SL.state = SL_State.EJECTED THEN
			// finished
			// reset own pointers
			SL.bIdx := 0;
			SL.wIdx := 0;
			SL.currW := TC.nullW;
			// reset fin
			fin := FALSE;
			SL.state := SL_State.WAITING_FOR_W;
			step := 1;
		END_IF
END_CASE
                    
END_ACTION

ACTION Init_active:
                      (*
Copyright (c) 2019 Manuel Goester, Michael Witt, Klaus Kammerer
Institute of Databases and Information Systems, Ulm University, Germany

Permission is hereby granted, free of charge, to any person obtaining a copy 
of this software and associated documentation files (the "Software"), to deal 
in the Software without restriction, including without limitation the rights 
to use, copy, modify, merge, publish, distribute, sublicense, and/or sell 
copies of the Software, and to permit persons to whom the Software is 
furnished to do so, subject to the following conditions:

The above copyright notice and this permission notice shall be included in 
all copies or substantial portions of the Software.

THE SOFTWARE IS PROVIDED "AS IS", WITHOUT WARRANTY OF ANY KIND, EXPRESS OR 
IMPLIED, INCLUDING BUT NOT LIMITED TO THE WARRANTIES OF MERCHANTABILITY, 
FITNESS FOR A PARTICULAR PURPOSE AND NONINFRINGEMENT. IN NO EVENT SHALL THE 
AUTHORS OR COPYRIGHT HOLDERS BE LIABLE FOR ANY CLAIM, DAMAGES OR OTHER 
LIABILITY, WHETHER IN AN ACTION OF CONTRACT, TORT OR OTHERWISE, ARISING FROM, 
OUT OF OR IN CONNECTION WITH THE SOFTWARE OR THE USE OR OTHER DEALINGS 
IN THE SOFTWARE.
*)
SL.state := SL_State.WAITING_FOR_W;
step := 1;
                    
END_ACTION
END_PROGRAM

(* Moves HR to certain position Copyright (c) 2019 Manuel Goester, Michael Witt, Klaus Kammerer Institute of Databases and Information Systems, Ulm University, Germany Permission is hereby granted, free of charge, to any person obtaining a copy of this software and associated documentation files (the "Software"), to deal in the Software without restriction, including without limitation the rights to use, copy, modify, merge, publish, distribute, sublicense, and/or sell copies of the Software, and to permit persons to whom the Software is furnished to do so, subject to the following conditions: The above copyright notice and this permission notice shall be included in all copies or substantial portions of the Software. THE SOFTWARE IS PROVIDED "AS IS", WITHOUT WARRANTY OF ANY KIND, EXPRESS OR IMPLIED, INCLUDING BUT NOT LIMITED TO THE WARRANTIES OF MERCHANTABILITY, FITNESS FOR A PARTICULAR PURPOSE AND NONINFRINGEMENT. IN NO EVENT SHALL THE AUTHORS OR COPYRIGHT HOLDERS BE LIABLE FOR ANY CLAIM, DAMAGES OR OTHER LIABILITY, WHETHER IN AN ACTION OF CONTRACT, TORT OR OTHERWISE, ARISING FROM, OUT OF OR IN CONNECTION WITH THE SOFTWARE OR THE USE OR OTHER DEALINGS IN THE SOFTWARE. *)
FUNCTION_BLOCK HR_MOVE_TO_POS
  VAR_INPUT
    pos : RackPos;  (* the position where to go *)
    upOrDown : RackPos;  (* the upper (RackPos.UP) or lower (RackPos.DOWN) position at pos *)
  END_VAR
  VAR
    x : INT;
    y : INT;
    xFin : BOOL := FALSE;  (* finish flags *)
    yFin : BOOL := FALSE;
    fin : BOOL := FALSE;
    xAlreadyCounted : BOOL := FALSE;  (* true, if an impulse coming from the motor has been already counted *)
    yAlreadyCounted : BOOL := FALSE;
  END_VAR

                  fin := FALSE;

// choose x and y values dependent on the position
CASE pos OF
	RackPos.RACK_11:
		x := 292;
		IF upOrDown = RackPos.DOWN THEN
			y := 17;
		ELSIF upOrDown = RackPos.UP THEN
			y := 1;
		END_IF
	RackPos.RACK_12:
		x := 203;
		IF upOrDown = RackPos.DOWN THEN
			y := 17;
		ELSIF upOrDown = RackPos.UP THEN
			y := 1;
		END_IF
	RackPos.RACK_13:
		x := 114;
		IF upOrDown = RackPos.DOWN THEN
			y := 17;
		ELSIF upOrDown = RackPos.UP THEN
			y := 1;
		END_IF
	RackPos.RACK_21:
		x := 292;
		IF upOrDown = RackPos.DOWN THEN
			y := 70;
		ELSIF upOrDown = RackPos.UP THEN
			y := 54;
		END_IF
	RackPos.RACK_22:
		x := 203;
		IF upOrDown = RackPos.DOWN THEN
			y := 70;
		ELSIF upOrDown = RackPos.UP THEN
			y := 54;
		END_IF
	RackPos.RACK_23:
		x := 114;
		IF upOrDown = RackPos.DOWN THEN
			y := 70;
		ELSIF upOrDown = RackPos.UP THEN
			y := 54;
		END_IF
	RackPos.RACK_31:
		x := 292;
		IF upOrDown = RackPos.DOWN THEN
			y := 129;
		ELSIF upOrDown = RackPos.UP THEN
			y := 113;
		END_IF
	RackPos.RACK_32:
		x := 203;
		IF upOrDown = RackPos.DOWN THEN
			y := 129;
		ELSIF upOrDown = RackPos.UP THEN
			y := 113;
		END_IF
	RackPos.RACK_33:
		x := 114;
		IF upOrDown = RackPos.DOWN THEN
			y := 129;
		ELSIF upOrDown = RackPos.UP THEN
			y := 113;
		END_IF
	RackPos.CONVEYOR:
		x := 0;
		IF upOrDown = RackPos.DOWN THEN
			y := 112;
		ELSIF upOrDown = RackPos.UP THEN
			y := 96;
		END_IF
END_CASE;

// to handle negative counter values
IF HR.cX < 0 THEN
	HR.cX := 0;
END_IF
IF HR.cY < 0 THEN
	HR.cY := 0;
END_IF

// X AXIS
IF HR.cX = x THEN
	// if counter reached demanded position, we're done
	HR.mHorizontalRight := FALSE;
	HR.mHorizontalLeft := FALSE;
	xFin := TRUE;
ELSE
	// SAVETY FIRST: HR does not move in x direction if cantilever is not driven back
	IF NOT(HR.sCBack) THEN
		HR.mCBackward := TRUE;
	ELSE
		HR.mCBackward := FALSE;
		xFin := FALSE;
		IF HR.cX < x AND NOT(xFin) THEN
			HR.mHorizontalLeft := TRUE;
			HR.mHorizontalRight := FALSE;
			IF HR.encHorizontal AND NOT(xAlreadyCounted) THEN
				HR.cX := HR.cX + 1;
				xAlreadyCounted := TRUE;
			ELSIF NOT(HR.encHorizontal) THEN
				xAlreadyCounted := FALSE;
			END_IF
		ELSIF HR.cX > x AND NOT(xFin) THEN
			HR.mHorizontalRight := TRUE;
			HR.mHorizontalLeft := FALSE;
			IF HR.encHorizontal AND NOT(xAlreadyCounted) THEN
				HR.cX := HR.cX - 1;
				xAlreadyCounted := TRUE;
			ELSIF NOT(HR.encHorizontal) THEN
				xAlreadyCounted := FALSE;
			END_IF
		END_IF
	END_IF
END_IF




// Y AXIS
IF HR.cY = y THEN
	// if counter reached demanded position, we're done
	HR.mVerticalUp := FALSE;
	HR.mVerticalDown := FALSE;
	yFin := TRUE;
ELSE
	yFin := FALSE;
	IF HR.cY < y AND NOT(yFin) THEN
		HR.mVerticalDown := TRUE;
		HR.mVerticalUp := FALSE;
		IF HR.encVertical AND NOT(yAlreadyCounted) THEN
			HR.cY := HR.cY + 1;
			yAlreadyCounted := TRUE;
		ELSIF NOT(HR.encVertical) THEN
			yAlreadyCounted := FALSE;
		END_IF
	ELSIF HR.cY > y AND NOT(yFin) THEN
		HR.mVerticalUp := TRUE;
		HR.mVerticalDown := FALSE;
		IF HR.encVertical AND NOT(yAlreadyCounted) THEN
			HR.cY := HR.cY - 1;
			yAlreadyCounted := TRUE;
		ELSIF NOT(HR.encVertical) THEN
			yAlreadyCounted := FALSE;
		END_IF
	END_IF
END_IF

// if x and y axis are finsihed, we're done
IF xFin AND yFin THEN
	xFin := FALSE;
	yFin := FALSE;
	fin := TRUE;
	RETURN;
END_IF
                
END_FUNCTION_BLOCK

(* HR takes a workpiece out of rack and brings it to conveyor Copyright (c) 2019 Manuel Goester, Michael Witt, Klaus Kammerer Institute of Databases and Information Systems, Ulm University, Germany Permission is hereby granted, free of charge, to any person obtaining a copy of this software and associated documentation files (the "Software"), to deal in the Software without restriction, including without limitation the rights to use, copy, modify, merge, publish, distribute, sublicense, and/or sell copies of the Software, and to permit persons to whom the Software is furnished to do so, subject to the following conditions: The above copyright notice and this permission notice shall be included in all copies or substantial portions of the Software. THE SOFTWARE IS PROVIDED "AS IS", WITHOUT WARRANTY OF ANY KIND, EXPRESS OR IMPLIED, INCLUDING BUT NOT LIMITED TO THE WARRANTIES OF MERCHANTABILITY, FITNESS FOR A PARTICULAR PURPOSE AND NONINFRINGEMENT. IN NO EVENT SHALL THE AUTHORS OR COPYRIGHT HOLDERS BE LIABLE FOR ANY CLAIM, DAMAGES OR OTHER LIABILITY, WHETHER IN AN ACTION OF CONTRACT, TORT OR OTHERWISE, ARISING FROM, OUT OF OR IN CONNECTION WITH THE SOFTWARE OR THE USE OR OTHER DEALINGS IN THE SOFTWARE. *)
FUNCTION_BLOCK HR_GET_W
  VAR_INPUT
    w : Workpiece;  (* the workpiece *)
  END_VAR
  VAR
    hr_move : HR_MOVE;
    hr_move_to_pos : HR_MOVE_TO_POS;
    hr_take_w : HR_TAKE_W;
    hr_put_w_on_conveyor : HR_PUT_W_ON_CONVEYOR;
    step : INT := 1;
    fin : BOOL := FALSE;
    stepFin : BOOL := FALSE;
  END_VAR

                  CASE step OF
	1: 	// to rack
		fin := FALSE;
		hr_move_to_pos(pos := w.startPos, upOrDown := RackPos.DOWN);
		stepFin := hr_move_to_pos.fin; 
		IF stepFin THEN
			step := step + 1;
			stepFin := FALSE;
		END_IF
	2:	// take w from rack
		hr_take_w(w := w);
		stepFin := hr_take_w.fin;
		IF stepFin THEN
			step := step + 1;
			stepFin := FALSE;
		END_IF
	3:	// to conveyor
		hr_move_to_pos(pos := RackPos.CONVEYOR, upOrDown := RackPos.UP);
		stepFin := hr_move_to_pos.fin;	
		IF stepFin THEN
			step := step + 1;
			stepFin := FALSE;
		END_IF
	
	4:	// finished
		fin := TRUE;
		step := 1;
		stepFin := FALSE;
END_CASE
                
END_FUNCTION_BLOCK

(* HR puts down a workpiece into rack or at conveyor Copyright (c) 2019 Manuel Goester, Michael Witt, Klaus Kammerer Institute of Databases and Information Systems, Ulm University, Germany Permission is hereby granted, free of charge, to any person obtaining a copy of this software and associated documentation files (the "Software"), to deal in the Software without restriction, including without limitation the rights to use, copy, modify, merge, publish, distribute, sublicense, and/or sell copies of the Software, and to permit persons to whom the Software is furnished to do so, subject to the following conditions: The above copyright notice and this permission notice shall be included in all copies or substantial portions of the Software. THE SOFTWARE IS PROVIDED "AS IS", WITHOUT WARRANTY OF ANY KIND, EXPRESS OR IMPLIED, INCLUDING BUT NOT LIMITED TO THE WARRANTIES OF MERCHANTABILITY, FITNESS FOR A PARTICULAR PURPOSE AND NONINFRINGEMENT. IN NO EVENT SHALL THE AUTHORS OR COPYRIGHT HOLDERS BE LIABLE FOR ANY CLAIM, DAMAGES OR OTHER LIABILITY, WHETHER IN AN ACTION OF CONTRACT, TORT OR OTHERWISE, ARISING FROM, OUT OF OR IN CONNECTION WITH THE SOFTWARE OR THE USE OR OTHER DEALINGS IN THE SOFTWARE. *)
FUNCTION_BLOCK HR_PUT_W
  VAR
    step : INT := 1;
    hr_move : HR_MOVE;
    fin : BOOL := FALSE;
    stepFin : BOOL := FALSE;
  END_VAR

                  CASE step OF
	1:	// forward
		fin := FALSE;
		IF NOT(HR.sCFront) THEN
			HR.mCForward := TRUE;
		ELSE
			HR.mCForward := FALSE;
			step := step + 1;
		END_IF
	2:	// down
		hr_move(x := 0 , y := 16);
		stepFin := hr_move.fin;
		IF stepFin THEN
			step := step + 1;
			stepFin := FALSE;
		END_IF
	3:	// back
		IF NOT(HR.sCBack) THEN
			HR.mCBackward := TRUE;
		ELSE
			HR.mCBackward := FALSE;
			step := step + 1;
		END_IF
	4:	// finished
		fin := TRUE;
		step := 1;
END_CASE
                
END_FUNCTION_BLOCK

PROGRAM HR_SORTING_MODE
  VAR
    hr_switch_ws : HR_SWITCH_WS;
    fin : BOOL;
  END_VAR

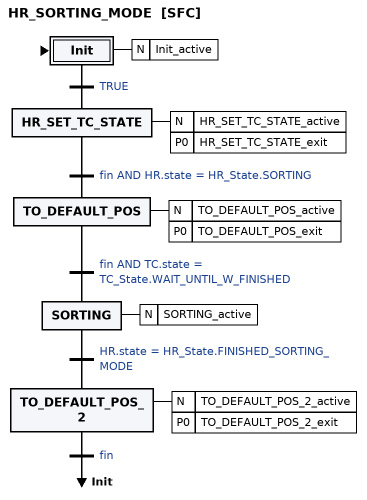
INITIAL_STEP Init:
  Init_active(N);
END_STEP
TRANSITION FROM Init TO HR_SET_TC_STATE
  := TRUE;
END_TRANSITION
STEP HR_SET_TC_STATE:
  HR_SET_TC_STATE_active(N);
  HR_SET_TC_STATE_exit(P0);
END_STEP
TRANSITION FROM HR_SET_TC_STATE TO TO_DEFAULT_POS
  := fin AND HR.state = HR_State.SORTING;
END_TRANSITION
STEP TO_DEFAULT_POS:
  TO_DEFAULT_POS_active(N);
  TO_DEFAULT_POS_exit(P0);
END_STEP
TRANSITION FROM TO_DEFAULT_POS TO SORTING
  := fin AND TC.state = TC_State.WAIT_UNTIL_W_FINISHED;
END_TRANSITION
STEP SORTING:
  SORTING_active(N);
END_STEP
TRANSITION FROM SORTING TO TO_DEFAULT_POS_2
  := HR.state = HR_State.FINISHED_SORTING_MODE;
END_TRANSITION
STEP TO_DEFAULT_POS_2:
  TO_DEFAULT_POS_2_active(N);
  TO_DEFAULT_POS_2_exit(P0);
END_STEP
TRANSITION FROM TO_DEFAULT_POS_2 TO Init
  := fin;
END_TRANSITION

ACTION SORTING_active:
                      (*
Copyright (c) 2019 Manuel Goester, Michael Witt, Klaus Kammerer
Institute of Databases and Information Systems, Ulm University, Germany

Permission is hereby granted, free of charge, to any person obtaining a copy 
of this software and associated documentation files (the "Software"), to deal 
in the Software without restriction, including without limitation the rights 
to use, copy, modify, merge, publish, distribute, sublicense, and/or sell 
copies of the Software, and to permit persons to whom the Software is 
furnished to do so, subject to the following conditions:

The above copyright notice and this permission notice shall be included in 
all copies or substantial portions of the Software.

THE SOFTWARE IS PROVIDED "AS IS", WITHOUT WARRANTY OF ANY KIND, EXPRESS OR 
IMPLIED, INCLUDING BUT NOT LIMITED TO THE WARRANTIES OF MERCHANTABILITY, 
FITNESS FOR A PARTICULAR PURPOSE AND NONINFRINGEMENT. IN NO EVENT SHALL THE 
AUTHORS OR COPYRIGHT HOLDERS BE LIABLE FOR ANY CLAIM, DAMAGES OR OTHER 
LIABILITY, WHETHER IN AN ACTION OF CONTRACT, TORT OR OTHERWISE, ARISING FROM, 
OUT OF OR IN CONNECTION WITH THE SOFTWARE OR THE USE OR OTHER DEALINGS 
IN THE SOFTWARE.
*)
IF NOT(fin) THEN
	hr_switch_ws(w1 := TC.batchJobQueue.batchJobs[TC.currBatchJobIdx].workpieces[TC.batchJobQueue.batchJobs[TC.currBatchJobIdx].nextNotProcessedIdx], w2 := TC.batchJobQueue.batchJobs[TC.currBatchJobIdx].workpieces[TC.batchJobQueue.batchJobs[TC.currBatchJobIdx].nextNotProcessedIdx+1]);
	fin := hr_switch_ws.fin;
ELSE
	// sorting finished
	fin := FALSE;
	HR.state := HR_State.FINISHED_SORTING_MODE;
END_IF

                    
END_ACTION

ACTION TO_DEFAULT_POS_exit:
                      (*
Copyright (c) 2019 Manuel Goester, Michael Witt, Klaus Kammerer
Institute of Databases and Information Systems, Ulm University, Germany

Permission is hereby granted, free of charge, to any person obtaining a copy 
of this software and associated documentation files (the "Software"), to deal 
in the Software without restriction, including without limitation the rights 
to use, copy, modify, merge, publish, distribute, sublicense, and/or sell 
copies of the Software, and to permit persons to whom the Software is 
furnished to do so, subject to the following conditions:

The above copyright notice and this permission notice shall be included in 
all copies or substantial portions of the Software.

THE SOFTWARE IS PROVIDED "AS IS", WITHOUT WARRANTY OF ANY KIND, EXPRESS OR 
IMPLIED, INCLUDING BUT NOT LIMITED TO THE WARRANTIES OF MERCHANTABILITY, 
FITNESS FOR A PARTICULAR PURPOSE AND NONINFRINGEMENT. IN NO EVENT SHALL THE 
AUTHORS OR COPYRIGHT HOLDERS BE LIABLE FOR ANY CLAIM, DAMAGES OR OTHER 
LIABILITY, WHETHER IN AN ACTION OF CONTRACT, TORT OR OTHERWISE, ARISING FROM, 
OUT OF OR IN CONNECTION WITH THE SOFTWARE OR THE USE OR OTHER DEALINGS 
IN THE SOFTWARE.
*)
fin := FALSE;
                    
END_ACTION

ACTION TO_DEFAULT_POS_active:
                      (*
Copyright (c) 2019 Manuel Goester, Michael Witt, Klaus Kammerer
Institute of Databases and Information Systems, Ulm University, Germany

Permission is hereby granted, free of charge, to any person obtaining a copy 
of this software and associated documentation files (the "Software"), to deal 
in the Software without restriction, including without limitation the rights 
to use, copy, modify, merge, publish, distribute, sublicense, and/or sell 
copies of the Software, and to permit persons to whom the Software is 
furnished to do so, subject to the following conditions:

The above copyright notice and this permission notice shall be included in 
all copies or substantial portions of the Software.

THE SOFTWARE IS PROVIDED "AS IS", WITHOUT WARRANTY OF ANY KIND, EXPRESS OR 
IMPLIED, INCLUDING BUT NOT LIMITED TO THE WARRANTIES OF MERCHANTABILITY, 
FITNESS FOR A PARTICULAR PURPOSE AND NONINFRINGEMENT. IN NO EVENT SHALL THE 
AUTHORS OR COPYRIGHT HOLDERS BE LIABLE FOR ANY CLAIM, DAMAGES OR OTHER 
LIABILITY, WHETHER IN AN ACTION OF CONTRACT, TORT OR OTHERWISE, ARISING FROM, 
OUT OF OR IN CONNECTION WITH THE SOFTWARE OR THE USE OR OTHER DEALINGS 
IN THE SOFTWARE.
*)
// get HR to its default position
IF HR.sCBack = FALSE THEN
	HR.mCBackward := TRUE;
ELSE 
	HR.mCBackward := FALSE;
	// set tower vertical position to max UP as well as horizontal position max RIGHT
	IF HR.sHorizontal = FALSE THEN
		HR.mHorizontalRight := TRUE;
	ELSE
		HR.mHorizontalRight := FALSE;
		HR.cX := 0;
	END_IF
	
	IF HR.sVertical = FALSE THEN
		HR.mVerticalUp := TRUE;
	ELSE
		HR.mVerticalUp := FALSE;
		HR.cY := 0;
	END_IF
END_IF

IF HR.sHorizontal AND HR.sVertical AND HR.sCBack THEN
	// finished
	fin := TRUE;
END_IF
                    
END_ACTION

ACTION Init_active:
                      
                    
END_ACTION

ACTION HR_SET_TC_STATE_active:
                      (*
Copyright (c) 2019 Manuel Goester, Michael Witt, Klaus Kammerer
Institute of Databases and Information Systems, Ulm University, Germany

Permission is hereby granted, free of charge, to any person obtaining a copy 
of this software and associated documentation files (the "Software"), to deal 
in the Software without restriction, including without limitation the rights 
to use, copy, modify, merge, publish, distribute, sublicense, and/or sell 
copies of the Software, and to permit persons to whom the Software is 
furnished to do so, subject to the following conditions:

The above copyright notice and this permission notice shall be included in 
all copies or substantial portions of the Software.

THE SOFTWARE IS PROVIDED "AS IS", WITHOUT WARRANTY OF ANY KIND, EXPRESS OR 
IMPLIED, INCLUDING BUT NOT LIMITED TO THE WARRANTIES OF MERCHANTABILITY, 
FITNESS FOR A PARTICULAR PURPOSE AND NONINFRINGEMENT. IN NO EVENT SHALL THE 
AUTHORS OR COPYRIGHT HOLDERS BE LIABLE FOR ANY CLAIM, DAMAGES OR OTHER 
LIABILITY, WHETHER IN AN ACTION OF CONTRACT, TORT OR OTHERWISE, ARISING FROM, 
OUT OF OR IN CONNECTION WITH THE SOFTWARE OR THE USE OR OTHER DEALINGS 
IN THE SOFTWARE.
*)
IF NOT(fin) THEN
	IF TC.state = TC_State.W_LOADED THEN
		TC.state := TC_State.WAIT_UNTIL_W_FINISHED;
		fin := TRUE;
	ELSE
		// load a new workpiece
		TC.state := TC_State.LOAD_NEXT_W;
	END_IF
END_IF

                    
END_ACTION

ACTION HR_SET_TC_STATE_exit:
                      (*
Copyright (c) 2019 Manuel Goester, Michael Witt, Klaus Kammerer
Institute of Databases and Information Systems, Ulm University, Germany

Permission is hereby granted, free of charge, to any person obtaining a copy 
of this software and associated documentation files (the "Software"), to deal 
in the Software without restriction, including without limitation the rights 
to use, copy, modify, merge, publish, distribute, sublicense, and/or sell 
copies of the Software, and to permit persons to whom the Software is 
furnished to do so, subject to the following conditions:

The above copyright notice and this permission notice shall be included in 
all copies or substantial portions of the Software.

THE SOFTWARE IS PROVIDED "AS IS", WITHOUT WARRANTY OF ANY KIND, EXPRESS OR 
IMPLIED, INCLUDING BUT NOT LIMITED TO THE WARRANTIES OF MERCHANTABILITY, 
FITNESS FOR A PARTICULAR PURPOSE AND NONINFRINGEMENT. IN NO EVENT SHALL THE 
AUTHORS OR COPYRIGHT HOLDERS BE LIABLE FOR ANY CLAIM, DAMAGES OR OTHER 
LIABILITY, WHETHER IN AN ACTION OF CONTRACT, TORT OR OTHERWISE, ARISING FROM, 
OUT OF OR IN CONNECTION WITH THE SOFTWARE OR THE USE OR OTHER DEALINGS 
IN THE SOFTWARE.
*)
fin := FALSE;
                    
END_ACTION

ACTION TO_DEFAULT_POS_2_exit:
                      (*
Copyright (c) 2019 Manuel Goester, Michael Witt, Klaus Kammerer
Institute of Databases and Information Systems, Ulm University, Germany

